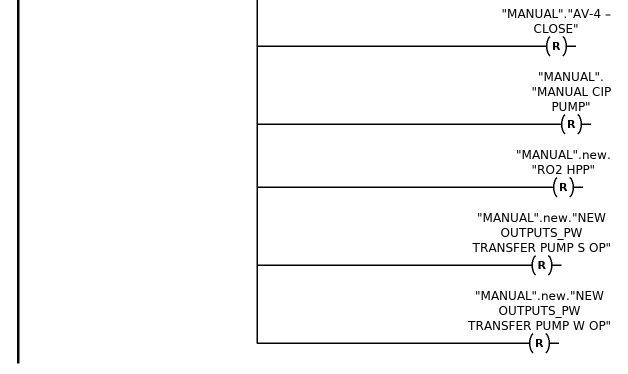
   RUNG wire#powerrail
      Contact( "AlwaysTRUE" )
      wire#w1
      { S7_Templates := "SrcType := Int" } NE_Contact(in1 := "Mode Select"."MFG MODE".BUFFER, in2 := 2)
      wire#w2
      R_Coil( "MANUAL"."MGF FEED PUMP WORKING" )
   END_RUNG
   RUNG wire#w1
      Contact( "INTERLOCK".ERROR )
   END_RUNG wire#w2
   RUNG wire#w2
      R_Coil( "MANUAL"."MFG FEED PUMP STANDBY" )
   END_RUNG
   RUNG wire#w2
      R_Coil( "MANUAL"."RO FEED PUMP WORKING" )
   END_RUNG
   RUNG wire#w2
      R_Coil( "MANUAL"."RO FEED PUMP STANDBY" )
   END_RUNG
   RUNG wire#w2
      R_Coil( "MANUAL"."RO HPP PUMP WORKING" )
   END_RUNG
   RUNG wire#w2
      R_Coil( "MANUAL"."RO HPP PUMP STANDBY" )
   END_RUNG
   RUNG wire#w2
      R_Coil( "MANUAL"."SMBS AGT-1" )
   END_RUNG
   RUNG wire#w2
      R_Coil( "MANUAL"."SALT TANK AGT-2" )
   END_RUNG
   RUNG wire#w2
      R_Coil( "MANUAL"."RO SMBS AGT-3" )
   END_RUNG
   RUNG wire#w2
      R_Coil( "MANUAL"."DP-1" )
   END_RUNG
   RUNG wire#w2
      R_Coil( "MANUAL"."DP-2" )
   END_RUNG
   RUNG wire#w2
      R_Coil( "MANUAL"."DP-3" )
   END_RUNG
   RUNG wire#w2
      R_Coil( "MANUAL"."DP-4" )
   END_RUNG
   RUNG wire#w2
      R_Coil( "MANUAL"."DP-5" )
   END_RUNG
   RUNG wire#w2
      R_Coil( "MANUAL"."DP-6" )
   END_RUNG
   RUNG wire#w2
      R_Coil( "MANUAL"."UV-1-DO" )
   END_RUNG
   RUNG wire#w2
      R_Coil( "MANUAL"."UV-2-DO" )
   END_RUNG
   RUNG wire#w2
      R_Coil( "MANUAL".HOOTER )
   END_RUNG
   RUNG wire#w2
      R_Coil( "MANUAL"."PSFV-1 – OPEN" )
   END_RUNG
   RUNG wire#w2
      R_Coil( "MANUAL"."PSFV-1 – CLOSE" )
   END_RUNG
   RUNG wire#w2
      R_Coil( "MANUAL"."PSFV-2 – OPEN" )
   END_RUNG
   RUNG wire#w2
      R_Coil( "MANUAL"."PSFV-2 – CLOSE" )
   END_RUNG
   RUNG wire#w2
      R_Coil( "MANUAL"."PSFV-3 – OPEN" )
   END_RUNG
   RUNG wire#w2
      R_Coil( "MANUAL"."PSFV-3 – CLOSE" )
   END_RUNG
   RUNG wire#w2
      R_Coil( "MANUAL"."PSFV-4 – OPEN" )
   END_RUNG
   RUNG wire#w2
      R_Coil( "MANUAL"."PSFV-4 – CLOSE" )
   END_RUNG
   RUNG wire#w2
      R_Coil( "MANUAL"."PSFV-5 – OPEN" )
   END_RUNG
   RUNG wire#w2
      R_Coil( "MANUAL"."PSFV-5 – CLOSE" )
   END_RUNG
   RUNG wire#w2
      R_Coil( "MANUAL"."PSFV-6 – OPEN" )
   END_RUNG
   RUNG wire#w2
      R_Coil( "MANUAL"."PSFV-6 – CLOSE" )
   END_RUNG
   RUNG wire#w2
      R_Coil( "MANUAL"."ACFV-1 – OPEN" )
   END_RUNG
   RUNG wire#w2
      R_Coil( "MANUAL"."ACFV-1 – CLOSE" )
   END_RUNG
   RUNG wire#w2
      R_Coil( "MANUAL"."ACFV-2 – OPEN" )
   END_RUNG
   RUNG wire#w2
      R_Coil( "MANUAL"."ACFV-2 – CLOSE" )
   END_RUNG
   RUNG wire#w2
      R_Coil( "MANUAL"."ACFV-3 – OPEN" )
   END_RUNG
   RUNG wire#w2
      R_Coil( "MANUAL"."ACFV-3 – CLOSE" )
   END_RUNG
   RUNG wire#w2
      R_Coil( "MANUAL"."ACFV-4 – OPEN" )
   END_RUNG
   RUNG wire#w2
      R_Coil( "MANUAL"."ACFV-4 - CLOSE" )
   END_RUNG
   RUNG wire#w2
      R_Coil( "MANUAL"."ACFV-5 – OPEN" )
   END_RUNG
   RUNG wire#w2
      R_Coil( "MANUAL"."ACFV-5 – CLOSE" )
   END_RUNG
   RUNG wire#w2
      R_Coil( "MANUAL"."ACFV-6 – OPEN" )
   END_RUNG
   RUNG wire#w2
      R_Coil( "MANUAL"."ACFV-6 – CLOSE" )
   END_RUNG
   RUNG wire#w2
      R_Coil( "MANUAL"."SFV-1 – OPEN" )
   END_RUNG
   RUNG wire#w2
      R_Coil( "MANUAL"."SFV-1 – CLOSE" )
   END_RUNG
   RUNG wire#w2
      R_Coil( "MANUAL"."SFV-2 – OPEN" )
   END_RUNG
   RUNG wire#w2
      R_Coil( "MANUAL"."SFV-2 – CLOSE" )
   END_RUNG
   RUNG wire#w2
      R_Coil( "MANUAL"."SFV-3 – OPEN" )
   END_RUNG
   RUNG wire#w2
      R_Coil( "MANUAL"."SFV-3 – CLOSE" )
   END_RUNG
   RUNG wire#w2
      R_Coil( "MANUAL"."SFV-4 – OPEN" )
   END_RUNG
   RUNG wire#w2
      R_Coil( "MANUAL"."SFV-4 – CLOSE" )
   END_RUNG
   RUNG wire#w2
      R_Coil( "MANUAL"."SFV-5 – OPEN" )
   END_RUNG
   RUNG wire#w2
      R_Coil( "MANUAL"."SFV-5 – CLOSE" )
   END_RUNG
   RUNG wire#w2
      R_Coil( "MANUAL"."SFV-6 – OPEN" )
   END_RUNG
   RUNG wire#w2
      R_Coil( "MANUAL"."SFV-6 – CLOSE" )
   END_RUNG
   RUNG wire#w2
      R_Coil( "MANUAL"."SFV-7 – OPEN" )
   END_RUNG
   RUNG wire#w2
      R_Coil( "MANUAL"."SFV-7 – CLOSE" )
   END_RUNG
   RUNG wire#w2
      R_Coil( "MANUAL"."SFV-8 – OPEN" )
   END_RUNG
   RUNG wire#w2
      R_Coil( "MANUAL"."SFV-8 – CLOSE" )
   END_RUNG
   RUNG wire#w2
      R_Coil( "MANUAL"."AV-1 – OPEN" )
   END_RUNG
   RUNG wire#w2
      R_Coil( "MANUAL"."AV-1 – CLOSE" )
   END_RUNG
   RUNG wire#w2
      R_Coil( "MANUAL"."AV-2 – OPEN" )
   END_RUNG
   RUNG wire#w2
      R_Coil( "MANUAL"."AV-2 – CLOSE" )
   END_RUNG
   RUNG wire#w2
      R_Coil( "MANUAL"."AV-3 – OPEN" )
   END_RUNG
   RUNG wire#w2
      R_Coil( "MANUAL"."AV-3 – CLOSE" )
   END_RUNG
   RUNG wire#w2
      R_Coil( "MANUAL"."AV-4 – OPEN" )
   END_RUNG
   RUNG wire#w2
      R_Coil( "MANUAL"."AV-4 – CLOSE" )
   END_RUNG
   RUNG wire#w2
      R_Coil( "MANUAL"."MANUAL CIP PUMP" )
   END_RUNG
   RUNG wire#w2
      R_Coil( "MANUAL".new."RO2 HPP" )
   END_RUNG
   RUNG wire#w2
      R_Coil( "MANUAL".new."NEW OUTPUTS_PW TRANSFER PUMP S OP" )
   END_RUNG
   RUNG wire#w2
      R_Coil( "MANUAL".new."NEW OUTPUTS_PW TRANSFER PUMP W OP" )
   END_RUNG
   // the same network as SCL:
   IF "AlwaysTRUE" AND (("Mode Select"."MFG MODE".BUFFER <> 2) OR "INTERLOCK".ERROR) THEN
       "MANUAL"."MGF FEED PUMP WORKING" := FALSE;
       "MANUAL"."MFG FEED PUMP STANDBY" := FALSE;
       "MANUAL"."RO FEED PUMP WORKING" := FALSE;
       "MANUAL"."RO FEED PUMP STANDBY" := FALSE;
       "MANUAL"."RO HPP PUMP WORKING" := FALSE;
       "MANUAL"."RO HPP PUMP STANDBY" := FALSE;
       "MANUAL"."SMBS AGT-1" := FALSE;
       "MANUAL"."SALT TANK AGT-2" := FALSE;
       "MANUAL"."RO SMBS AGT-3" := FALSE;
       "MANUAL"."DP-1" := FALSE;
       "MANUAL"."DP-2" := FALSE;
       "MANUAL"."DP-3" := FALSE;
       "MANUAL"."DP-4" := FALSE;
       "MANUAL"."DP-5" := FALSE;
       "MANUAL"."DP-6" := FALSE;
       "MANUAL"."UV-1-DO" := FALSE;
       "MANUAL"."UV-2-DO" := FALSE;
       "MANUAL".HOOTER := FALSE;
       "MANUAL"."PSFV-1 – OPEN" := FALSE;
       "MANUAL"."PSFV-1 – CLOSE" := FALSE;
       "MANUAL"."PSFV-2 – OPEN" := FALSE;
       "MANUAL"."PSFV-2 – CLOSE" := FALSE;
       "MANUAL"."PSFV-3 – OPEN" := FALSE;
       "MANUAL"."PSFV-3 – CLOSE" := FALSE;
       "MANUAL"."PSFV-4 – OPEN" := FALSE;
       "MANUAL"."PSFV-4 – CLOSE" := FALSE;
       "MANUAL"."PSFV-5 – OPEN" := FALSE;
       "MANUAL"."PSFV-5 – CLOSE" := FALSE;
       "MANUAL"."PSFV-6 – OPEN" := FALSE;
       "MANUAL"."PSFV-6 – CLOSE" := FALSE;
       "MANUAL"."ACFV-1 – OPEN" := FALSE;
       "MANUAL"."ACFV-1 – CLOSE" := FALSE;
       "MANUAL"."ACFV-2 – OPEN" := FALSE;
       "MANUAL"."ACFV-2 – CLOSE" := FALSE;
       "MANUAL"."ACFV-3 – OPEN" := FALSE;
       "MANUAL"."ACFV-3 – CLOSE" := FALSE;
       "MANUAL"."ACFV-4 – OPEN" := FALSE;
       "MANUAL"."ACFV-4 - CLOSE" := FALSE;
       "MANUAL"."ACFV-5 – OPEN" := FALSE;
       "MANUAL"."ACFV-5 – CLOSE" := FALSE;
       "MANUAL"."ACFV-6 – OPEN" := FALSE;
       "MANUAL"."ACFV-6 – CLOSE" := FALSE;
       "MANUAL"."SFV-1 – OPEN" := FALSE;
       "MANUAL"."SFV-1 – CLOSE" := FALSE;
       "MANUAL"."SFV-2 – OPEN" := FALSE;
       "MANUAL"."SFV-2 – CLOSE" := FALSE;
       "MANUAL"."SFV-3 – OPEN" := FALSE;
       "MANUAL"."SFV-3 – CLOSE" := FALSE;
       "MANUAL"."SFV-4 – OPEN" := FALSE;
       "MANUAL"."SFV-4 – CLOSE" := FALSE;
       "MANUAL"."SFV-5 – OPEN" := FALSE;
       "MANUAL"."SFV-5 – CLOSE" := FALSE;
       "MANUAL"."SFV-6 – OPEN" := FALSE;
       "MANUAL"."SFV-6 – CLOSE" := FALSE;
       "MANUAL"."SFV-7 – OPEN" := FALSE;
       "MANUAL"."SFV-7 – CLOSE" := FALSE;
       "MANUAL"."SFV-8 – OPEN" := FALSE;
       "MANUAL"."SFV-8 – CLOSE" := FALSE;
       "MANUAL"."AV-1 – OPEN" := FALSE;
       "MANUAL"."AV-1 – CLOSE" := FALSE;
       "MANUAL"."AV-2 – OPEN" := FALSE;
       "MANUAL"."AV-2 – CLOSE" := FALSE;
       "MANUAL"."AV-3 – OPEN" := FALSE;
       "MANUAL"."AV-3 – CLOSE" := FALSE;
       "MANUAL"."AV-4 – OPEN" := FALSE;
       "MANUAL"."AV-4 – CLOSE" := FALSE;
       "MANUAL"."MANUAL CIP PUMP" := FALSE;
       "MANUAL".new."RO2 HPP" := FALSE;
       "MANUAL".new."NEW OUTPUTS_PW TRANSFER PUMP S OP" := FALSE;
       "MANUAL".new."NEW OUTPUTS_PW TRANSFER PUMP W OP" := FALSE;
   END_IF;
END_REGION

REGION Network 3: TRANSFER PUMP WORKING & STANDBY
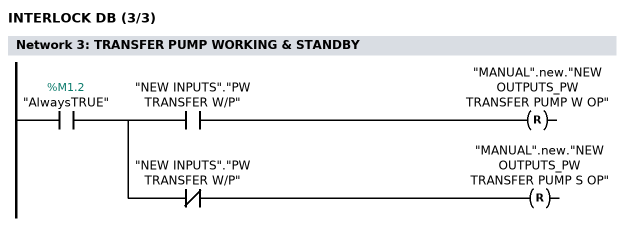
   RUNG wire#powerrail
      Contact( "AlwaysTRUE" )
      wire#w1
      Contact( "NEW INPUTS"."PW TRANSFER W/P" )
      R_Coil( "MANUAL".new."NEW OUTPUTS_PW TRANSFER PUMP W OP" )
   END_RUNG
   RUNG wire#w1
      I_Contact( "NEW INPUTS"."PW TRANSFER W/P" )
      R_Coil( "MANUAL".new."NEW OUTPUTS_PW TRANSFER PUMP S OP" )
   END_RUNG
   // the same network as SCL:
   IF "AlwaysTRUE" AND "NEW INPUTS"."PW TRANSFER W/P" THEN
       "MANUAL".new."NEW OUTPUTS_PW TRANSFER PUMP W OP" := FALSE;
   END_IF;
   IF "AlwaysTRUE" AND NOT "NEW INPUTS"."PW TRANSFER W/P" THEN
       "MANUAL".new."NEW OUTPUTS_PW TRANSFER PUMP S OP" := FALSE;
   END_IF;
END_REGION
END_FUNCTION

FUNCTION "SCALING" : Void   // FC3, LAD
{ S7_Optimized_Access := 'TRUE' }
// stored: SetENOAutomatically false
BEGIN

REGION Network 1: LT-1
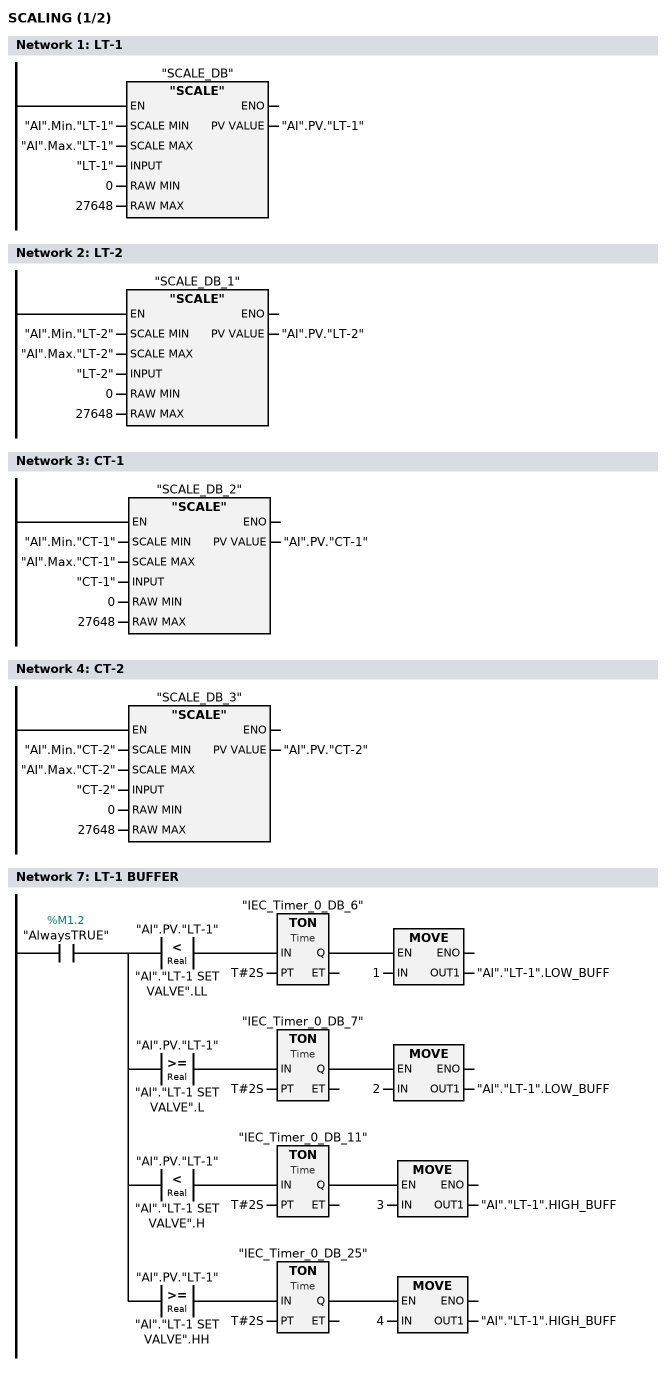
   RUNG wire#powerrail
      "SCALE_DB"("SCALE MIN" := "AI".Min."LT-1", "SCALE MAX" := "AI".Max."LT-1", INPUT := "LT-1", "RAW MIN" := 0, "RAW MAX" := 27648, "PV VALUE" => "AI".PV."LT-1")
   END_RUNG
   // the same network as SCL:
   "SCALE_DB"("SCALE MIN" := "AI".Min."LT-1",   // "SCALE"
              "SCALE MAX" := "AI".Max."LT-1",
              INPUT := "LT-1",
              "RAW MIN" := 0,
              "RAW MAX" := 27648,
              "PV VALUE" => "AI".PV."LT-1");
END_REGION

REGION Network 2: LT-2
   RUNG wire#powerrail
      "SCALE_DB_1"("SCALE MIN" := "AI".Min."LT-2", "SCALE MAX" := "AI".Max."LT-2", INPUT := "LT-2", "RAW MIN" := 0, "RAW MAX" := 27648, "PV VALUE" => "AI".PV."LT-2")
   END_RUNG
   // the same network as SCL:
   "SCALE_DB_1"("SCALE MIN" := "AI".Min."LT-2",   // "SCALE"
                "SCALE MAX" := "AI".Max."LT-2",
                INPUT := "LT-2",
                "RAW MIN" := 0,
                "RAW MAX" := 27648,
                "PV VALUE" => "AI".PV."LT-2");
END_REGION

REGION Network 3: CT-1
   RUNG wire#powerrail
      "SCALE_DB_2"("SCALE MIN" := "AI".Min."CT-1", "SCALE MAX" := "AI".Max."CT-1", INPUT := "CT-1", "RAW MIN" := 0, "RAW MAX" := 27648, "PV VALUE" => "AI".PV."CT-1")
   END_RUNG
   // the same network as SCL:
   "SCALE_DB_2"("SCALE MIN" := "AI".Min."CT-1",   // "SCALE"
                "SCALE MAX" := "AI".Max."CT-1",
                INPUT := "CT-1",
                "RAW MIN" := 0,
                "RAW MAX" := 27648,
                "PV VALUE" => "AI".PV."CT-1");
END_REGION

REGION Network 4: CT-2
   RUNG wire#powerrail
      "SCALE_DB_3"("SCALE MIN" := "AI".Min."CT-2", "SCALE MAX" := "AI".Max."CT-2", INPUT := "CT-2", "RAW MIN" := 0, "RAW MAX" := 27648, "PV VALUE" => "AI".PV."CT-2")
   END_RUNG
   // the same network as SCL:
   "SCALE_DB_3"("SCALE MIN" := "AI".Min."CT-2",   // "SCALE"
                "SCALE MAX" := "AI".Max."CT-2",
                INPUT := "CT-2",
                "RAW MIN" := 0,
                "RAW MAX" := 27648,
                "PV VALUE" => "AI".PV."CT-2");
END_REGION

REGION Network 7: LT-1 BUFFER
   RUNG wire#powerrail
      Contact( "AlwaysTRUE" )
      wire#w1
      { S7_Templates := "SrcType := Real" } LT_Contact(in1 := "AI".PV."LT-1", in2 := "AI"."LT-1 SET VALVE".LL)
      { S7_Templates := "time_type := Time" } "IEC_Timer_0_DB_6".TON(pt := T#2S, et =>)
      Move(in := 1, out1 => "AI"."LT-1".LOW_BUFF)
   END_RUNG
   RUNG wire#w1
      { S7_Templates := "SrcType := Real" } GE_Contact(in1 := "AI".PV."LT-1", in2 := "AI"."LT-1 SET VALVE".L)
      { S7_Templates := "time_type := Time" } "IEC_Timer_0_DB_7".TON(pt := T#2S, et =>)
      Move(in := 2, out1 => "AI"."LT-1".LOW_BUFF)
   END_RUNG
   RUNG wire#w1
      { S7_Templates := "SrcType := Real" } LT_Contact(in1 := "AI".PV."LT-1", in2 := "AI"."LT-1 SET VALVE".H)
      { S7_Templates := "time_type := Time" } "IEC_Timer_0_DB_11".TON(pt := T#2S, et =>)
      Move(in := 3, out1 => "AI"."LT-1".HIGH_BUFF)
   END_RUNG
   RUNG wire#w1
      { S7_Templates := "SrcType := Real" } GE_Contact(in1 := "AI".PV."LT-1", in2 := "AI"."LT-1 SET VALVE".HH)
      { S7_Templates := "time_type := Time" } "IEC_Timer_0_DB_25".TON(pt := T#2S, et =>)
      Move(in := 4, out1 => "AI"."LT-1".HIGH_BUFF)
   END_RUNG
   // the same network as SCL:
   "IEC_Timer_0_DB_6".TON(IN := "AlwaysTRUE" AND ("AI".PV."LT-1" < "AI"."LT-1 SET VALVE".LL), PT := T#2S);
   IF "IEC_Timer_0_DB_6".Q THEN "AI"."LT-1".LOW_BUFF := 1; END_IF;
   "IEC_Timer_0_DB_7".TON(IN := "AlwaysTRUE" AND ("AI".PV."LT-1" >= "AI"."LT-1 SET VALVE".L), PT := T#2S);
   IF "IEC_Timer_0_DB_7".Q THEN "AI"."LT-1".LOW_BUFF := 2; END_IF;
   "IEC_Timer_0_DB_11".TON(IN := "AlwaysTRUE" AND ("AI".PV."LT-1" < "AI"."LT-1 SET VALVE".H), PT := T#2S);
   IF "IEC_Timer_0_DB_11".Q THEN "AI"."LT-1".HIGH_BUFF := 3; END_IF;
   "IEC_Timer_0_DB_25".TON(IN := "AlwaysTRUE" AND ("AI".PV."LT-1" >= "AI"."LT-1 SET VALVE".HH), PT := T#2S);
   IF "IEC_Timer_0_DB_25".Q THEN "AI"."LT-1".HIGH_BUFF := 4; END_IF;
END_REGION

REGION Network 8: LT-2 BUFFER
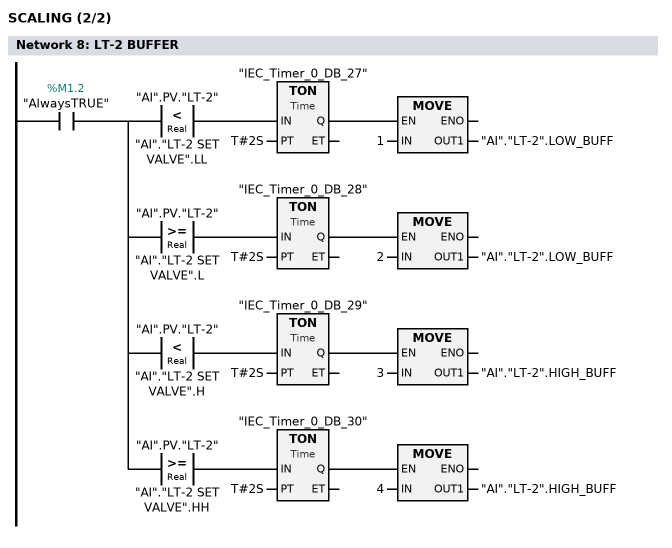
   RUNG wire#powerrail
      Contact( "AlwaysTRUE" )
      wire#w1
      { S7_Templates := "SrcType := Real" } LT_Contact(in1 := "AI".PV."LT-2", in2 := "AI"."LT-2 SET VALVE".LL)
      { S7_Templates := "time_type := Time" } "IEC_Timer_0_DB_27".TON(pt := T#2S, et =>)
      Move(in := 1, out1 => "AI"."LT-2".LOW_BUFF)
   END_RUNG
   RUNG wire#w1
      { S7_Templates := "SrcType := Real" } GE_Contact(in1 := "AI".PV."LT-2", in2 := "AI"."LT-2 SET VALVE".L)
      { S7_Templates := "time_type := Time" } "IEC_Timer_0_DB_28".TON(pt := T#2S, et =>)
      Move(in := 2, out1 => "AI"."LT-2".LOW_BUFF)
   END_RUNG
   RUNG wire#w1
      { S7_Templates := "SrcType := Real" } LT_Contact(in1 := "AI".PV."LT-2", in2 := "AI"."LT-2 SET VALVE".H)
      { S7_Templates := "time_type := Time" } "IEC_Timer_0_DB_29".TON(pt := T#2S, et =>)
      Move(in := 3, out1 => "AI"."LT-2".HIGH_BUFF)
   END_RUNG
   RUNG wire#w1
      { S7_Templates := "SrcType := Real" } GE_Contact(in1 := "AI".PV."LT-2", in2 := "AI"."LT-2 SET VALVE".HH)
      { S7_Templates := "time_type := Time" } "IEC_Timer_0_DB_30".TON(pt := T#2S, et =>)
      Move(in := 4, out1 => "AI"."LT-2".HIGH_BUFF)
   END_RUNG
   // the same network as SCL:
   "IEC_Timer_0_DB_27".TON(IN := "AlwaysTRUE" AND ("AI".PV."LT-2" < "AI"."LT-2 SET VALVE".LL), PT := T#2S);
   IF "IEC_Timer_0_DB_27".Q THEN "AI"."LT-2".LOW_BUFF := 1; END_IF;
   "IEC_Timer_0_DB_28".TON(IN := "AlwaysTRUE" AND ("AI".PV."LT-2" >= "AI"."LT-2 SET VALVE".L), PT := T#2S);
   IF "IEC_Timer_0_DB_28".Q THEN "AI"."LT-2".LOW_BUFF := 2; END_IF;
   "IEC_Timer_0_DB_29".TON(IN := "AlwaysTRUE" AND ("AI".PV."LT-2" < "AI"."LT-2 SET VALVE".H), PT := T#2S);
   IF "IEC_Timer_0_DB_29".Q THEN "AI"."LT-2".HIGH_BUFF := 3; END_IF;
   "IEC_Timer_0_DB_30".TON(IN := "AlwaysTRUE" AND ("AI".PV."LT-2" >= "AI"."LT-2 SET VALVE".HH), PT := T#2S);
   IF "IEC_Timer_0_DB_30".Q THEN "AI"."LT-2".HIGH_BUFF := 4; END_IF;
END_REGION
END_FUNCTION

FUNCTION_BLOCK "SCALE"   // FB4, LAD
{ S7_Optimized_Access := 'TRUE' }
// stored: MemoryReserve 100, SetENOAutomatically false
   VAR_INPUT
      "SCALE MIN" : Real;
      "SCALE MAX" : Real;
      INPUT : Int;
      "RAW MIN" : Int;
      "RAW MAX" : Int;
   END_VAR
   VAR_OUTPUT
      "PV VALUE" : Real;
   END_VAR
   VAR_TEMP
      NORMX : Real;
   END_VAR
BEGIN

REGION Network 1
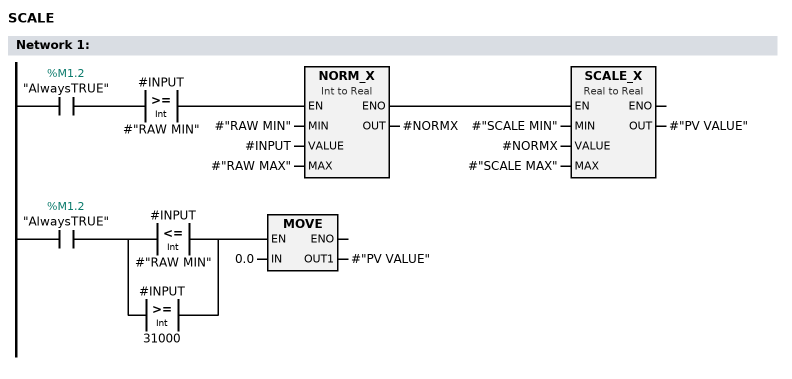
   RUNG wire#powerrail
      Contact( "AlwaysTRUE" )
      { S7_Templates := "SrcType := Int" } GE_Contact(in1 := #INPUT, in2 := #"RAW MIN")
      { S7_Templates := "[SrcType := Int, DestType := Real]" } Normalize(min := #"RAW MIN", value := #INPUT, max := #"RAW MAX", out => #NORMX)
      { S7_Templates := "[SrcType := Real, DestType := Real]" } Scale(min := #"SCALE MIN", value := #NORMX, max := #"SCALE MAX", out => #"PV VALUE")
   END_RUNG
   RUNG wire#powerrail
      Contact( "AlwaysTRUE" )
      wire#w1
      { S7_Templates := "SrcType := Int" } LE_Contact(in1 := #INPUT, in2 := #"RAW MIN")
      wire#w2
      Move(in := 0.0, out1 => #"PV VALUE")
   END_RUNG
   RUNG wire#w1
      { S7_Templates := "SrcType := Int" } GE_Contact(in1 := #INPUT, in2 := 31000)
   END_RUNG wire#w2
   // the same network as SCL:
   IF "AlwaysTRUE" AND (#INPUT >= #"RAW MIN") THEN
       #NORMX := NORM_X(MIN := #"RAW MIN", VALUE := #INPUT, MAX := #"RAW MAX");
       #"PV VALUE" := SCALE_X(MIN := #"SCALE MIN", VALUE := #NORMX, MAX := #"SCALE MAX");
   END_IF;
   IF "AlwaysTRUE" AND ((#INPUT <= #"RAW MIN") OR (#INPUT >= 31000)) THEN #"PV VALUE" := 0.0; END_IF;
END_REGION
END_FUNCTION_BLOCK

FUNCTION "ALARMS" : Void   // FC16, LAD
{ S7_Optimized_Access := 'TRUE' }
// stored: SetENOAutomatically false
   VAR_TEMP   // added for the SCL form of the ladder/FBD networks
      _w1 : Bool;
   END_VAR
BEGIN

REGION Network 1: EMG ALARM
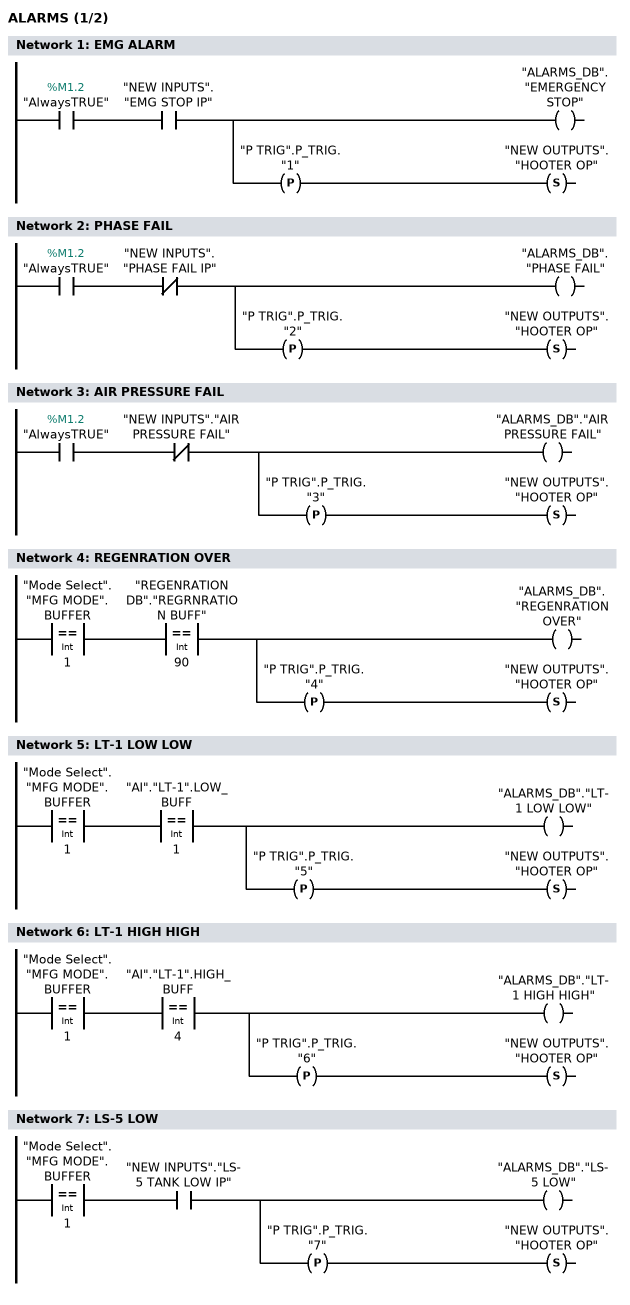
   RUNG wire#powerrail
      Contact( "AlwaysTRUE" )
      Contact( "NEW INPUTS"."EMG STOP IP" )
      wire#w1
      Coil( "ALARMS_DB"."EMERGENCY STOP" )
   END_RUNG
   RUNG wire#w1
      P_Trig( "P TRIG".P_TRIG."1" )
      S_Coil( "NEW OUTPUTS"."HOOTER OP" )
   END_RUNG
   // the same network as SCL:
   "ALARMS_DB"."EMERGENCY STOP" := "AlwaysTRUE" AND "NEW INPUTS"."EMG STOP IP";
   #_w1 := "ALARMS_DB"."EMERGENCY STOP" AND NOT "P TRIG".P_TRIG."1";   // rising edge
   "P TRIG".P_TRIG."1" := "ALARMS_DB"."EMERGENCY STOP";
   IF #_w1 THEN "NEW OUTPUTS"."HOOTER OP" := TRUE; END_IF;
END_REGION

REGION Network 2: PHASE FAIL
   RUNG wire#powerrail
      Contact( "AlwaysTRUE" )
      I_Contact( "NEW INPUTS"."PHASE FAIL IP" )
      wire#w1
      Coil( "ALARMS_DB"."PHASE FAIL" )
   END_RUNG
   RUNG wire#w1
      P_Trig( "P TRIG".P_TRIG."2" )
      S_Coil( "NEW OUTPUTS"."HOOTER OP" )
   END_RUNG
   // the same network as SCL:
   "ALARMS_DB"."PHASE FAIL" := "AlwaysTRUE" AND NOT "NEW INPUTS"."PHASE FAIL IP";
   #_w1 := "ALARMS_DB"."PHASE FAIL" AND NOT "P TRIG".P_TRIG."2";   // rising edge
   "P TRIG".P_TRIG."2" := "ALARMS_DB"."PHASE FAIL";
   IF #_w1 THEN "NEW OUTPUTS"."HOOTER OP" := TRUE; END_IF;
END_REGION

REGION Network 3: AIR PRESSURE FAIL
   RUNG wire#powerrail
      Contact( "AlwaysTRUE" )
      I_Contact( "NEW INPUTS"."AIR PRESSURE FAIL" )
      wire#w1
      Coil( "ALARMS_DB"."AIR PRESSURE FAIL" )
   END_RUNG
   RUNG wire#w1
      P_Trig( "P TRIG".P_TRIG."3" )
      S_Coil( "NEW OUTPUTS"."HOOTER OP" )
   END_RUNG
   // the same network as SCL:
   "ALARMS_DB"."AIR PRESSURE FAIL" := "AlwaysTRUE" AND NOT "NEW INPUTS"."AIR PRESSURE FAIL";
   #_w1 := "ALARMS_DB"."AIR PRESSURE FAIL" AND NOT "P TRIG".P_TRIG."3";   // rising edge
   "P TRIG".P_TRIG."3" := "ALARMS_DB"."AIR PRESSURE FAIL";
   IF #_w1 THEN "NEW OUTPUTS"."HOOTER OP" := TRUE; END_IF;
END_REGION

REGION Network 4: REGENRATION OVER
   RUNG wire#powerrail
      { S7_Templates := "SrcType := Int" } EQ_Contact(in1 := "Mode Select"."MFG MODE".BUFFER, in2 := 1)
      { S7_Templates := "SrcType := Int" } EQ_Contact(in1 := "REGENRATION DB"."REGRNRATION BUFF", in2 := 90)
      wire#w1
      Coil( "ALARMS_DB"."REGENRATION OVER" )
   END_RUNG
   RUNG wire#w1
      P_Trig( "P TRIG".P_TRIG."4" )
      S_Coil( "NEW OUTPUTS"."HOOTER OP" )
   END_RUNG
   // the same network as SCL:
   "ALARMS_DB"."REGENRATION OVER" := ("Mode Select"."MFG MODE".BUFFER = 1) AND ("REGENRATION DB"."REGRNRATION BUFF" = 90);
   #_w1 := "ALARMS_DB"."REGENRATION OVER" AND NOT "P TRIG".P_TRIG."4";   // rising edge
   "P TRIG".P_TRIG."4" := "ALARMS_DB"."REGENRATION OVER";
   IF #_w1 THEN "NEW OUTPUTS"."HOOTER OP" := TRUE; END_IF;
END_REGION

REGION Network 5: LT-1 LOW LOW
   RUNG wire#powerrail
      { S7_Templates := "SrcType := Int" } EQ_Contact(in1 := "Mode Select"."MFG MODE".BUFFER, in2 := 1)
      { S7_Templates := "SrcType := Int" } EQ_Contact(in1 := "AI"."LT-1".LOW_BUFF, in2 := 1)
      wire#w1
      Coil( "ALARMS_DB"."LT-1 LOW LOW" )
   END_RUNG
   RUNG wire#w1
      P_Trig( "P TRIG".P_TRIG."5" )
      S_Coil( "NEW OUTPUTS"."HOOTER OP" )
   END_RUNG
   // the same network as SCL:
   "ALARMS_DB"."LT-1 LOW LOW" := ("Mode Select"."MFG MODE".BUFFER = 1) AND ("AI"."LT-1".LOW_BUFF = 1);
   #_w1 := "ALARMS_DB"."LT-1 LOW LOW" AND NOT "P TRIG".P_TRIG."5";   // rising edge
   "P TRIG".P_TRIG."5" := "ALARMS_DB"."LT-1 LOW LOW";
   IF #_w1 THEN "NEW OUTPUTS"."HOOTER OP" := TRUE; END_IF;
END_REGION

REGION Network 6: LT-1 HIGH HIGH
   RUNG wire#powerrail
      { S7_Templates := "SrcType := Int" } EQ_Contact(in1 := "Mode Select"."MFG MODE".BUFFER, in2 := 1)
      { S7_Templates := "SrcType := Int" } EQ_Contact(in1 := "AI"."LT-1".HIGH_BUFF, in2 := 4)
      wire#w1
      Coil( "ALARMS_DB"."LT-1 HIGH HIGH" )
   END_RUNG
   RUNG wire#w1
      P_Trig( "P TRIG".P_TRIG."6" )
      S_Coil( "NEW OUTPUTS"."HOOTER OP" )
   END_RUNG
   // the same network as SCL:
   "ALARMS_DB"."LT-1 HIGH HIGH" := ("Mode Select"."MFG MODE".BUFFER = 1) AND ("AI"."LT-1".HIGH_BUFF = 4);
   #_w1 := "ALARMS_DB"."LT-1 HIGH HIGH" AND NOT "P TRIG".P_TRIG."6";   // rising edge
   "P TRIG".P_TRIG."6" := "ALARMS_DB"."LT-1 HIGH HIGH";
   IF #_w1 THEN "NEW OUTPUTS"."HOOTER OP" := TRUE; END_IF;
END_REGION

REGION Network 7: LS-5 LOW
   RUNG wire#powerrail
      { S7_Templates := "SrcType := Int" } EQ_Contact(in1 := "Mode Select"."MFG MODE".BUFFER, in2 := 1)
      Contact( "NEW INPUTS"."LS-5 TANK LOW IP" )
      wire#w1
      Coil( "ALARMS_DB"."LS-5 LOW" )
   END_RUNG
   RUNG wire#w1
      P_Trig( "P TRIG".P_TRIG."7" )
      S_Coil( "NEW OUTPUTS"."HOOTER OP" )
   END_RUNG
   // the same network as SCL:
   "ALARMS_DB"."LS-5 LOW" := ("Mode Select"."MFG MODE".BUFFER = 1) AND "NEW INPUTS"."LS-5 TANK LOW IP";
   #_w1 := "ALARMS_DB"."LS-5 LOW" AND NOT "P TRIG".P_TRIG."7";   // rising edge
   "P TRIG".P_TRIG."7" := "ALARMS_DB"."LS-5 LOW";
   IF #_w1 THEN "NEW OUTPUTS"."HOOTER OP" := TRUE; END_IF;
END_REGION

REGION Network 8: PS-1 LOW
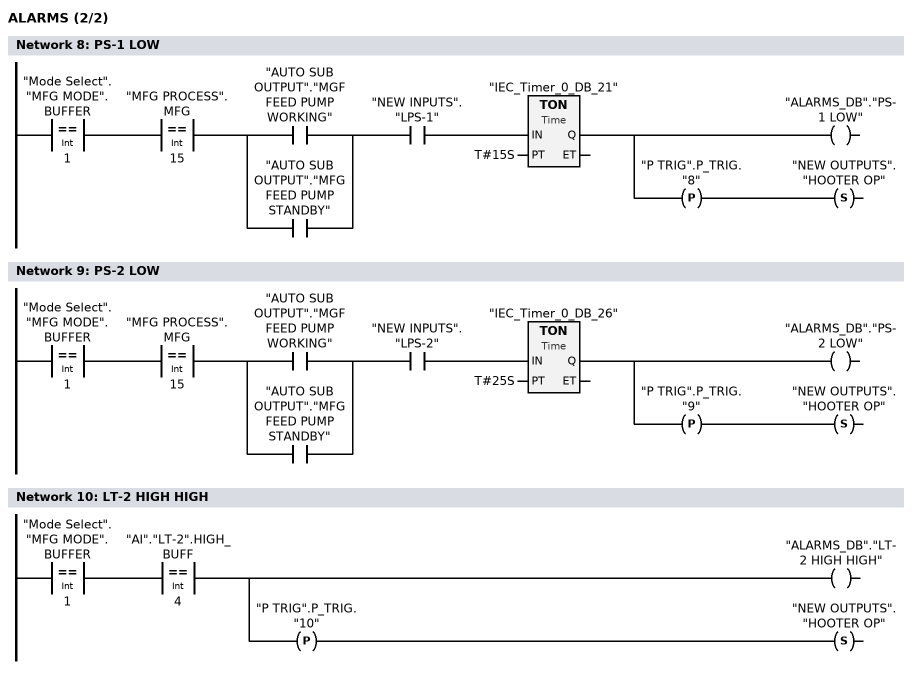
   RUNG wire#powerrail
      { S7_Templates := "SrcType := Int" } EQ_Contact(in1 := "Mode Select"."MFG MODE".BUFFER, in2 := 1)
      { S7_Templates := "SrcType := Int" } EQ_Contact(in1 := "MFG PROCESS".MFG, in2 := 15)
      wire#w1
      Contact( "AUTO SUB OUTPUT"."MGF FEED PUMP WORKING" )
      wire#w2
      Contact( "NEW INPUTS"."LPS-1" )
      { S7_Templates := "time_type := Time" } "IEC_Timer_0_DB_21".TON(pt := T#15S, et =>)
      wire#w3
      Coil( "ALARMS_DB"."PS-1 LOW" )
   END_RUNG
   RUNG wire#w1
      Contact( "AUTO SUB OUTPUT"."MFG FEED PUMP STANDBY" )
   END_RUNG wire#w2
   RUNG wire#w3
      P_Trig( "P TRIG".P_TRIG."8" )
      S_Coil( "NEW OUTPUTS"."HOOTER OP" )
   END_RUNG
   // the same network as SCL:
   "IEC_Timer_0_DB_21".TON(IN := ("Mode Select"."MFG MODE".BUFFER = 1) AND ("MFG PROCESS".MFG = 15) AND ("AUTO SUB OUTPUT"."MGF FEED PUMP WORKING" OR "AUTO SUB OUTPUT"."MFG FEED PUMP STANDBY") AND "NEW INPUTS"."LPS-1",
                           PT := T#15S);
   "ALARMS_DB"."PS-1 LOW" := "IEC_Timer_0_DB_21".Q;
   #_w1 := "IEC_Timer_0_DB_21".Q AND NOT "P TRIG".P_TRIG."8";   // rising edge
   "P TRIG".P_TRIG."8" := "IEC_Timer_0_DB_21".Q;
   IF #_w1 THEN "NEW OUTPUTS"."HOOTER OP" := TRUE; END_IF;
END_REGION

REGION Network 9: PS-2 LOW
   RUNG wire#powerrail
      { S7_Templates := "SrcType := Int" } EQ_Contact(in1 := "Mode Select"."MFG MODE".BUFFER, in2 := 1)
      { S7_Templates := "SrcType := Int" } EQ_Contact(in1 := "MFG PROCESS".MFG, in2 := 15)
      wire#w1
      Contact( "AUTO SUB OUTPUT"."MGF FEED PUMP WORKING" )
      wire#w2
      Contact( "NEW INPUTS"."LPS-2" )
      { S7_Templates := "time_type := Time" } "IEC_Timer_0_DB_26".TON(pt := T#25S, et =>)
      wire#w3
      Coil( "ALARMS_DB"."PS-2 LOW" )
   END_RUNG
   RUNG wire#w1
      Contact( "AUTO SUB OUTPUT"."MFG FEED PUMP STANDBY" )
   END_RUNG wire#w2
   RUNG wire#w3
      P_Trig( "P TRIG".P_TRIG."9" )
      S_Coil( "NEW OUTPUTS"."HOOTER OP" )
   END_RUNG
   // the same network as SCL:
   "IEC_Timer_0_DB_26".TON(IN := ("Mode Select"."MFG MODE".BUFFER = 1) AND ("MFG PROCESS".MFG = 15) AND ("AUTO SUB OUTPUT"."MGF FEED PUMP WORKING" OR "AUTO SUB OUTPUT"."MFG FEED PUMP STANDBY") AND "NEW INPUTS"."LPS-2",
                           PT := T#25S);
   "ALARMS_DB"."PS-2 LOW" := "IEC_Timer_0_DB_26".Q;
   #_w1 := "IEC_Timer_0_DB_26".Q AND NOT "P TRIG".P_TRIG."9";   // rising edge
   "P TRIG".P_TRIG."9" := "IEC_Timer_0_DB_26".Q;
   IF #_w1 THEN "NEW OUTPUTS"."HOOTER OP" := TRUE; END_IF;
END_REGION

REGION Network 10: LT-2 HIGH HIGH
   RUNG wire#powerrail
      { S7_Templates := "SrcType := Int" } EQ_Contact(in1 := "Mode Select"."MFG MODE".BUFFER, in2 := 1)
      { S7_Templates := "SrcType := Int" } EQ_Contact(in1 := "AI"."LT-2".HIGH_BUFF, in2 := 4)
      wire#w1
      Coil( "ALARMS_DB"."LT-2 HIGH HIGH" )
   END_RUNG
   RUNG wire#w1
      P_Trig( "P TRIG".P_TRIG."10" )
      S_Coil( "NEW OUTPUTS"."HOOTER OP" )
   END_RUNG
   // the same network as SCL:
   "ALARMS_DB"."LT-2 HIGH HIGH" := ("Mode Select"."MFG MODE".BUFFER = 1) AND ("AI"."LT-2".HIGH_BUFF = 4);
   #_w1 := "ALARMS_DB"."LT-2 HIGH HIGH" AND NOT "P TRIG".P_TRIG."10";   // rising edge
   "P TRIG".P_TRIG."10" := "ALARMS_DB"."LT-2 HIGH HIGH";
   IF #_w1 THEN "NEW OUTPUTS"."HOOTER OP" := TRUE; END_IF;
END_REGION
END_FUNCTION

FUNCTION "24 HOUR TIMER" : Void   // FC12, LAD
{ S7_Optimized_Access := 'TRUE' }
// stored: SetENOAutomatically false
   VAR_TEMP   // added for the SCL form of the ladder/FBD networks
      _w1 : Bool;
   END_VAR
BEGIN

REGION Network 1: 24 HOUR_TIMER
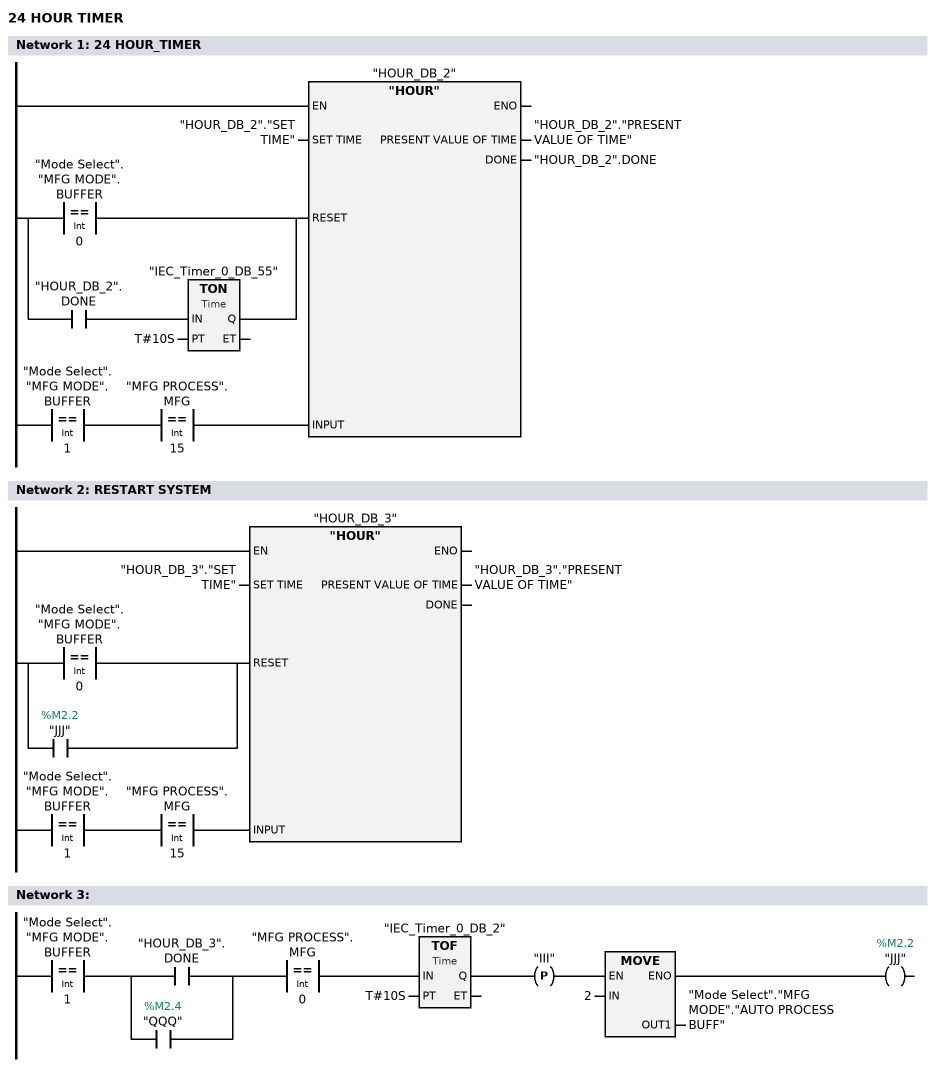
   RUNG wire#powerrail
      "HOUR_DB_2"(RESET := wire#w1, INPUT := wire#w2, "SET TIME" := "HOUR_DB_2"."SET TIME", "PRESENT VALUE OF TIME" => "HOUR_DB_2"."PRESENT VALUE OF TIME", DONE => "HOUR_DB_2".DONE)
   END_RUNG
   RUNG wire#powerrail
      { S7_Templates := "SrcType := Int" } EQ_Contact(in1 := "Mode Select"."MFG MODE".BUFFER, in2 := 0)
   END_RUNG wire#w1
   RUNG wire#powerrail
      Contact( "HOUR_DB_2".DONE )
      { S7_Templates := "time_type := Time" } "IEC_Timer_0_DB_55".TON(pt := T#10S, et =>)
   END_RUNG wire#w1
   RUNG wire#powerrail
      { S7_Templates := "SrcType := Int" } EQ_Contact(in1 := "Mode Select"."MFG MODE".BUFFER, in2 := 1)
      { S7_Templates := "SrcType := Int" } EQ_Contact(in1 := "MFG PROCESS".MFG, in2 := 15)
   END_RUNG wire#w2
   // the same network as SCL:
   "IEC_Timer_0_DB_55".TON(IN := "HOUR_DB_2".DONE, PT := T#10S);
   "HOUR_DB_2"("SET TIME" := "HOUR_DB_2"."SET TIME",   // "HOUR"
               RESET := ("Mode Select"."MFG MODE".BUFFER = 0) OR "IEC_Timer_0_DB_55".Q,
               INPUT := ("Mode Select"."MFG MODE".BUFFER = 1) AND ("MFG PROCESS".MFG = 15),
               "PRESENT VALUE OF TIME" => "HOUR_DB_2"."PRESENT VALUE OF TIME",
               DONE => "HOUR_DB_2".DONE);
END_REGION

REGION Network 2: RESTART SYSTEM
   RUNG wire#powerrail
      "HOUR_DB_3"(RESET := wire#w1, INPUT := wire#w2, "SET TIME" := "HOUR_DB_3"."SET TIME", "PRESENT VALUE OF TIME" => "HOUR_DB_3"."PRESENT VALUE OF TIME", DONE =>)
   END_RUNG
   RUNG wire#powerrail
      { S7_Templates := "SrcType := Int" } EQ_Contact(in1 := "Mode Select"."MFG MODE".BUFFER, in2 := 0)
   END_RUNG wire#w1
   RUNG wire#powerrail
      Contact( "JJJ" )
   END_RUNG wire#w1
   RUNG wire#powerrail
      { S7_Templates := "SrcType := Int" } EQ_Contact(in1 := "Mode Select"."MFG MODE".BUFFER, in2 := 1)
      { S7_Templates := "SrcType := Int" } EQ_Contact(in1 := "MFG PROCESS".MFG, in2 := 15)
   END_RUNG wire#w2
   // the same network as SCL:
   "HOUR_DB_3"("SET TIME" := "HOUR_DB_3"."SET TIME",   // "HOUR"
               RESET := ("Mode Select"."MFG MODE".BUFFER = 0) OR "JJJ",
               INPUT := ("Mode Select"."MFG MODE".BUFFER = 1) AND ("MFG PROCESS".MFG = 15),
               "PRESENT VALUE OF TIME" => "HOUR_DB_3"."PRESENT VALUE OF TIME");
END_REGION

REGION Network 3
   RUNG wire#powerrail
      { S7_Templates := "SrcType := Int" } EQ_Contact(in1 := "Mode Select"."MFG MODE".BUFFER, in2 := 1)
      wire#w1
      Contact( "HOUR_DB_3".DONE )
      wire#w2
      { S7_Templates := "SrcType := Int" } EQ_Contact(in1 := "MFG PROCESS".MFG, in2 := 0)
      { S7_Templates := "time_type := Time" } "IEC_Timer_0_DB_2".TOF(pt := T#10S, et =>)
      P_Trig( "III" )
      Move(in := 2, out1 => "Mode Select"."MFG MODE"."AUTO PROCESS BUFF")
      Coil( "JJJ" )
   END_RUNG
   RUNG wire#w1
      Contact( "QQQ" )
   END_RUNG wire#w2
   // the same network as SCL:
   "IEC_Timer_0_DB_2".TOF(IN := ("Mode Select"."MFG MODE".BUFFER = 1) AND ("HOUR_DB_3".DONE OR "QQQ") AND ("MFG PROCESS".MFG = 0),
                          PT := T#10S);
   #_w1 := "IEC_Timer_0_DB_2".Q AND NOT "III";   // rising edge
   "III" := "IEC_Timer_0_DB_2".Q;
   IF #_w1 THEN "Mode Select"."MFG MODE"."AUTO PROCESS BUFF" := 2; END_IF;
   "JJJ" := #_w1;
END_REGION
END_FUNCTION

FUNCTION_BLOCK "HOUR"   // FB2, LAD
{ S7_Optimized_Access := 'TRUE' }
// stored: MemoryReserve 100, SetENOAutomatically false
   VAR_INPUT
      "SET TIME" : Int;
      RESET : Bool;
      INPUT : Bool;
   END_VAR
   VAR_OUTPUT
      "PRESENT VALUE OF TIME" : Int;
      DONE : Bool;
   END_VAR
   VAR
      "TIMER 1" { S7_SetPoint := 'True'} : IEC_TIMER;
   END_VAR
   VAR RETAIN
      "COUNTER1 2" { S7_SetPoint := 'True'} : IEC_COUNTER;
      "COUNTER1 1" { S7_SetPoint := 'True'} : IEC_COUNTER;
   END_VAR
   VAR
      BIT { ExternalAccessible := 'False'; ExternalVisible := 'False'; ExternalWritable := 'False'} : Bool;
   END_VAR
   VAR_TEMP   // added for the SCL form of the ladder/FBD networks
      _w1 : Bool;
      _w2 : Bool;
   END_VAR
BEGIN

REGION Network 1
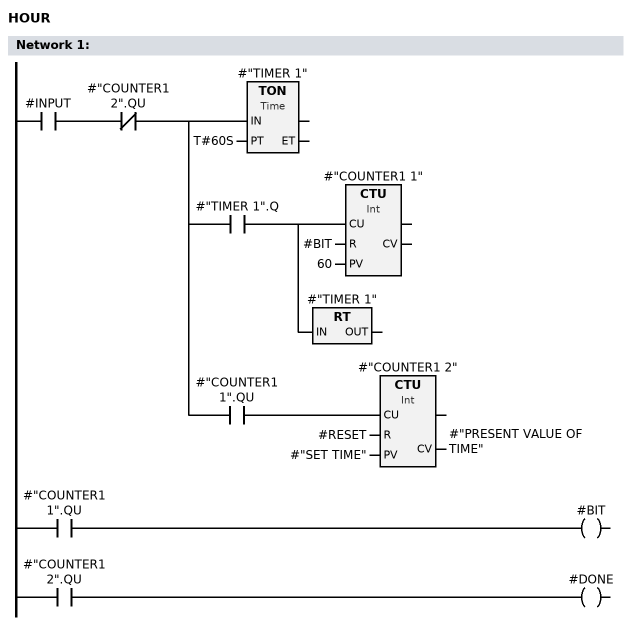
   RUNG wire#powerrail
      Contact( #INPUT )
      I_Contact( #"COUNTER1 2".QU )
      wire#w1
      { S7_Templates := "time_type := Time" } #"TIMER 1".TON(pt := T#60S, et =>)
   END_RUNG
   RUNG wire#w1
      Contact( #"TIMER 1".Q )
      wire#w2
      { S7_Templates := "value_type := Int" } #"COUNTER1 1".CTU(r := #BIT, pv := 60, cv =>)
   END_RUNG
   RUNG wire#w2
      RT_Coil( #"TIMER 1" )
   END_RUNG
   RUNG wire#w1
      Contact( #"COUNTER1 1".QU )
      { S7_Templates := "value_type := Int" } #"COUNTER1 2".CTU(r := #RESET, pv := #"SET TIME", cv => #"PRESENT VALUE OF TIME")
   END_RUNG
   RUNG wire#powerrail
      Contact( #"COUNTER1 1".QU )
      Coil( #BIT )
   END_RUNG
   RUNG wire#powerrail
      Contact( #"COUNTER1 2".QU )
      Coil( #DONE )
   END_RUNG
   // the same network as SCL:
   #_w1 := #INPUT AND NOT #"COUNTER1 2".QU;
   #"TIMER 1".TON(IN := #_w1, PT := T#60S);
   #_w2 := #_w1 AND #"TIMER 1".Q;
   #"COUNTER1 1".CTU(CU := #_w2, R := #BIT, PV := 60);
   IF #_w2 THEN RESET_TIMER(#"TIMER 1"); END_IF;
   #"COUNTER1 2".CTU(CU := #_w1 AND #"COUNTER1 1".QU,
                     R := #RESET,
                     PV := #"SET TIME",
                     CV => #"PRESENT VALUE OF TIME");
   #BIT := #"COUNTER1 1".QU;
   #DONE := #"COUNTER1 2".QU;
END_REGION
END_FUNCTION_BLOCK

FUNCTION "mfg filtration LOGIC" : Void   // FC8, LAD
{ S7_Optimized_Access := 'TRUE' }
// stored: SetENOAutomatically false
   VAR_TEMP   // added for the SCL form of the ladder/FBD networks
      _w1 : Bool;
   END_VAR
BEGIN

REGION Network 1: MFG PROCESS START
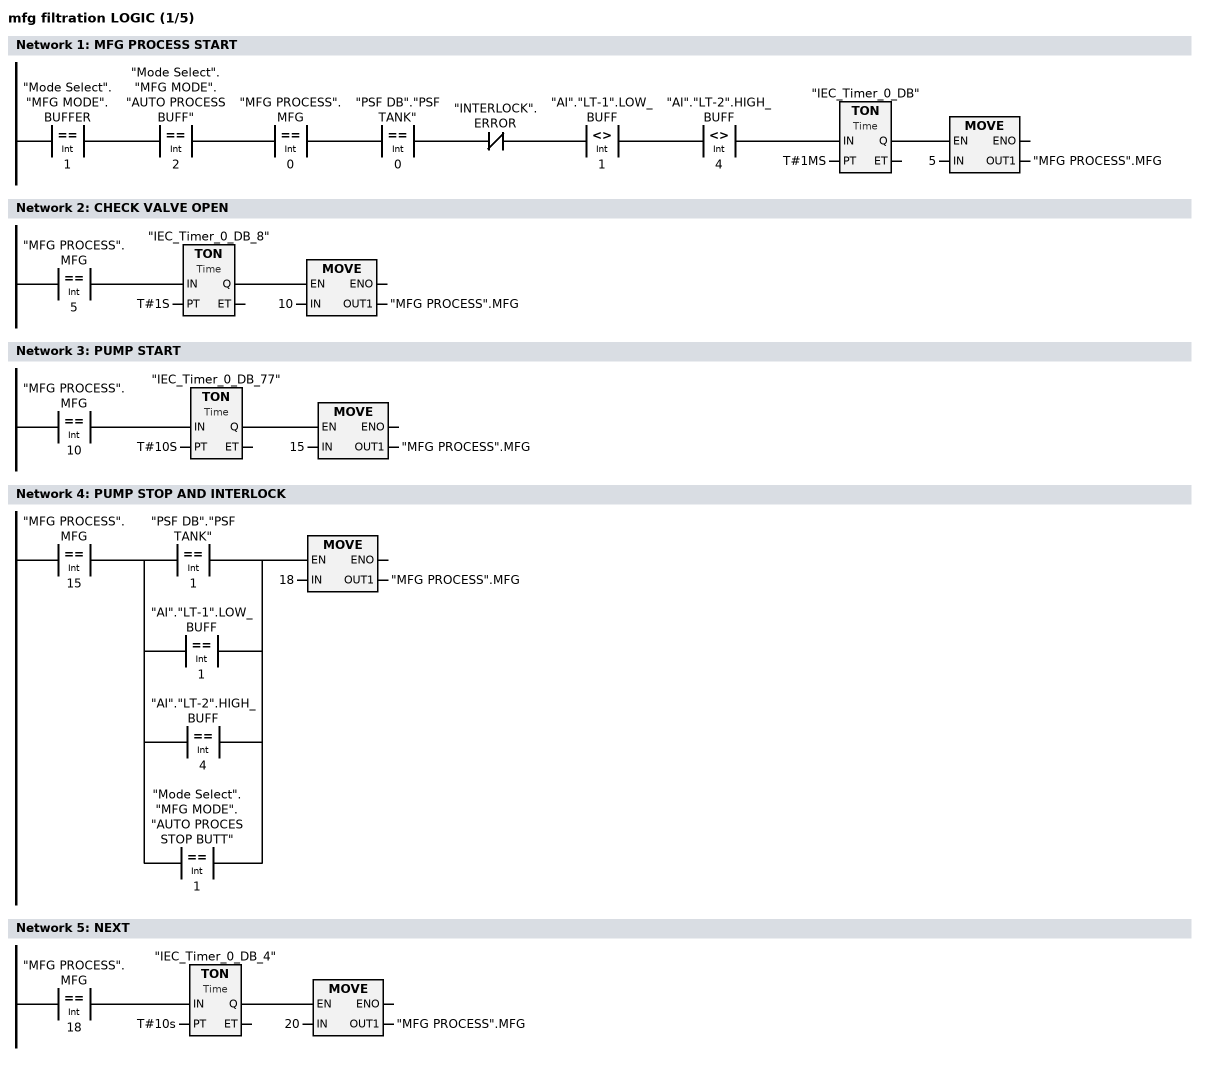
   RUNG wire#powerrail
      { S7_Templates := "SrcType := Int" } EQ_Contact(in1 := "Mode Select"."MFG MODE".BUFFER, in2 := 1)
      { S7_Templates := "SrcType := Int" } EQ_Contact(in1 := "Mode Select"."MFG MODE"."AUTO PROCESS BUFF", in2 := 2)
      { S7_Templates := "SrcType := Int" } EQ_Contact(in1 := "MFG PROCESS".MFG, in2 := 0)
      { S7_Templates := "SrcType := Int" } EQ_Contact(in1 := "PSF DB"."PSF TANK", in2 := 0)
      I_Contact( "INTERLOCK".ERROR )
      { S7_Templates := "SrcType := Int" } NE_Contact(in1 := "AI"."LT-1".LOW_BUFF, in2 := 1)
      { S7_Templates := "SrcType := Int" } NE_Contact(in1 := "AI"."LT-2".HIGH_BUFF, in2 := 4)
      { S7_Templates := "time_type := Time" } "IEC_Timer_0_DB".TON(pt := T#1MS, et =>)
      Move(in := 5, out1 => "MFG PROCESS".MFG)
   END_RUNG
   // the same network as SCL:
   "IEC_Timer_0_DB".TON(IN := ("Mode Select"."MFG MODE".BUFFER = 1) AND ("Mode Select"."MFG MODE"."AUTO PROCESS BUFF" = 2) AND ("MFG PROCESS".MFG = 0) AND ("PSF DB"."PSF TANK" = 0) AND NOT "INTERLOCK".ERROR AND ("AI"."LT-1".LOW_BUFF <> 1) AND ("AI"."LT-2".HIGH_BUFF <> 4),
                        PT := T#1MS);
   IF "IEC_Timer_0_DB".Q THEN "MFG PROCESS".MFG := 5; END_IF;
END_REGION

REGION Network 2: CHECK VALVE OPEN
   RUNG wire#powerrail
      { S7_Templates := "SrcType := Int" } EQ_Contact(in1 := "MFG PROCESS".MFG, in2 := 5)
      { S7_Templates := "time_type := Time" } "IEC_Timer_0_DB_8".TON(pt := T#1S, et =>)
      Move(in := 10, out1 => "MFG PROCESS".MFG)
   END_RUNG
   // the same network as SCL:
   "IEC_Timer_0_DB_8".TON(IN := "MFG PROCESS".MFG = 5, PT := T#1S);
   IF "IEC_Timer_0_DB_8".Q THEN "MFG PROCESS".MFG := 10; END_IF;
END_REGION

REGION Network 3: PUMP START
   RUNG wire#powerrail
      { S7_Templates := "SrcType := Int" } EQ_Contact(in1 := "MFG PROCESS".MFG, in2 := 10)
      { S7_Templates := "time_type := Time" } "IEC_Timer_0_DB_77".TON(pt := T#10S, et =>)
      Move(in := 15, out1 => "MFG PROCESS".MFG)
   END_RUNG
   // the same network as SCL:
   "IEC_Timer_0_DB_77".TON(IN := "MFG PROCESS".MFG = 10, PT := T#10S);
   IF "IEC_Timer_0_DB_77".Q THEN "MFG PROCESS".MFG := 15; END_IF;
END_REGION

REGION Network 4: PUMP STOP AND INTERLOCK
   RUNG wire#powerrail
      { S7_Templates := "SrcType := Int" } EQ_Contact(in1 := "MFG PROCESS".MFG, in2 := 15)
      wire#w1
      { S7_Templates := "SrcType := Int" } EQ_Contact(in1 := "PSF DB"."PSF TANK", in2 := 1)
      wire#w2
      Move(in := 18, out1 => "MFG PROCESS".MFG)
   END_RUNG
   RUNG wire#w1
      { S7_Templates := "SrcType := Int" } EQ_Contact(in1 := "AI"."LT-1".LOW_BUFF, in2 := 1)
   END_RUNG wire#w2
   RUNG wire#w1
      { S7_Templates := "SrcType := Int" } EQ_Contact(in1 := "AI"."LT-2".HIGH_BUFF, in2 := 4)
   END_RUNG wire#w2
   RUNG wire#w1
      { S7_Templates := "SrcType := Int" } EQ_Contact(in1 := "Mode Select"."MFG MODE"."AUTO PROCES STOP BUTT", in2 := 1)
   END_RUNG wire#w2
   // the same network as SCL:
   IF ("MFG PROCESS".MFG = 15) AND (("PSF DB"."PSF TANK" = 1) OR ("AI"."LT-1".LOW_BUFF = 1) OR ("AI"."LT-2".HIGH_BUFF = 4) OR ("Mode Select"."MFG MODE"."AUTO PROCES STOP BUTT" = 1)) THEN
       "MFG PROCESS".MFG := 18;
   END_IF;
END_REGION

REGION Network 5: NEXT
   RUNG wire#powerrail
      { S7_Templates := "SrcType := Int" } EQ_Contact(in1 := "MFG PROCESS".MFG, in2 := 18)
      { S7_Templates := "time_type := Time" } "IEC_Timer_0_DB_4".TON(pt := T#10s, et =>)
      Move(in := 20, out1 => "MFG PROCESS".MFG)
   END_RUNG
   // the same network as SCL:
   "IEC_Timer_0_DB_4".TON(IN := "MFG PROCESS".MFG = 18, PT := T#10s);
   IF "IEC_Timer_0_DB_4".Q THEN "MFG PROCESS".MFG := 20; END_IF;
END_REGION

REGION Network 6: MFG PROCESS OVER
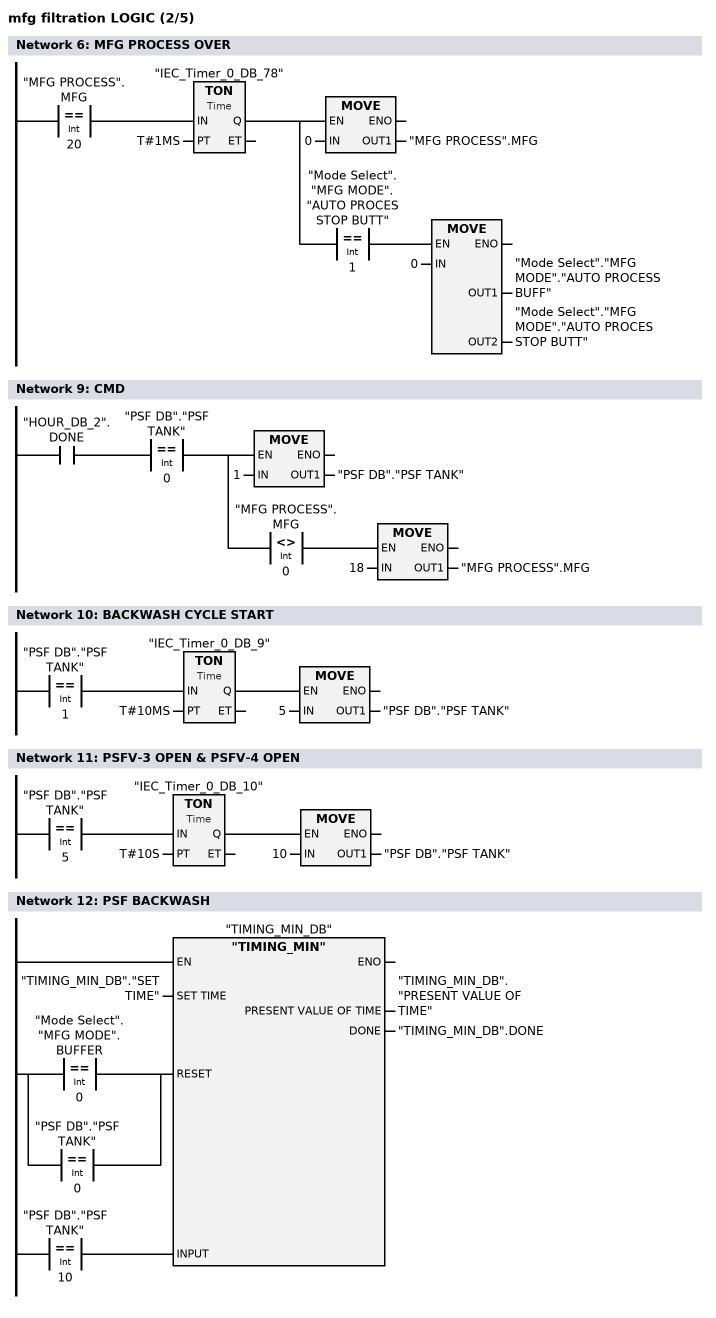
   RUNG wire#powerrail
      { S7_Templates := "SrcType := Int" } EQ_Contact(in1 := "MFG PROCESS".MFG, in2 := 20)
      { S7_Templates := "time_type := Time" } "IEC_Timer_0_DB_78".TON(pt := T#1MS, et =>)
      wire#w1
      Move(in := 0, out1 => "MFG PROCESS".MFG)
   END_RUNG
   RUNG wire#w1
      { S7_Templates := "SrcType := Int" } EQ_Contact(in1 := "Mode Select"."MFG MODE"."AUTO PROCES STOP BUTT", in2 := 1)
      Move(in := 0, out1 => "Mode Select"."MFG MODE"."AUTO PROCESS BUFF", out2 => "Mode Select"."MFG MODE"."AUTO PROCES STOP BUTT")
   END_RUNG
   // the same network as SCL:
   "IEC_Timer_0_DB_78".TON(IN := "MFG PROCESS".MFG = 20, PT := T#1MS);
   IF "IEC_Timer_0_DB_78".Q THEN "MFG PROCESS".MFG := 0; END_IF;
   IF "IEC_Timer_0_DB_78".Q AND ("Mode Select"."MFG MODE"."AUTO PROCES STOP BUTT" = 1) THEN
       "Mode Select"."MFG MODE"."AUTO PROCESS BUFF" := 0;
       "Mode Select"."MFG MODE"."AUTO PROCES STOP BUTT" := 0;
   END_IF;
END_REGION

REGION Network 9: CMD
   RUNG wire#powerrail
      Contact( "HOUR_DB_2".DONE )
      { S7_Templates := "SrcType := Int" } EQ_Contact(in1 := "PSF DB"."PSF TANK", in2 := 0)
      wire#w1
      Move(in := 1, out1 => "PSF DB"."PSF TANK")
   END_RUNG
   RUNG wire#w1
      { S7_Templates := "SrcType := Int" } NE_Contact(in1 := "MFG PROCESS".MFG, in2 := 0)
      Move(in := 18, out1 => "MFG PROCESS".MFG)
   END_RUNG
   // the same network as SCL:
   #_w1 := "HOUR_DB_2".DONE AND ("PSF DB"."PSF TANK" = 0);
   IF #_w1 THEN "PSF DB"."PSF TANK" := 1; END_IF;
   IF #_w1 AND ("MFG PROCESS".MFG <> 0) THEN "MFG PROCESS".MFG := 18; END_IF;
END_REGION

REGION Network 10: BACKWASH CYCLE START
   RUNG wire#powerrail
      { S7_Templates := "SrcType := Int" } EQ_Contact(in1 := "PSF DB"."PSF TANK", in2 := 1)
      { S7_Templates := "time_type := Time" } "IEC_Timer_0_DB_9".TON(pt := T#10MS, et =>)
      Move(in := 5, out1 => "PSF DB"."PSF TANK")
   END_RUNG
   // the same network as SCL:
   "IEC_Timer_0_DB_9".TON(IN := "PSF DB"."PSF TANK" = 1, PT := T#10MS);
   IF "IEC_Timer_0_DB_9".Q THEN "PSF DB"."PSF TANK" := 5; END_IF;
END_REGION

REGION Network 11: PSFV-3 OPEN & PSFV-4 OPEN
   RUNG wire#powerrail
      { S7_Templates := "SrcType := Int" } EQ_Contact(in1 := "PSF DB"."PSF TANK", in2 := 5)
      { S7_Templates := "time_type := Time" } "IEC_Timer_0_DB_10".TON(pt := T#10S, et =>)
      Move(in := 10, out1 => "PSF DB"."PSF TANK")
   END_RUNG
   // the same network as SCL:
   "IEC_Timer_0_DB_10".TON(IN := "PSF DB"."PSF TANK" = 5, PT := T#10S);
   IF "IEC_Timer_0_DB_10".Q THEN "PSF DB"."PSF TANK" := 10; END_IF;
END_REGION

REGION Network 12: PSF BACKWASH
   RUNG wire#powerrail
      "TIMING_MIN_DB"(RESET := wire#w1, INPUT := wire#w2, "SET TIME" := "TIMING_MIN_DB"."SET TIME", "PRESENT VALUE OF TIME" => "TIMING_MIN_DB"."PRESENT VALUE OF TIME", DONE => "TIMING_MIN_DB".DONE)
   END_RUNG
   RUNG wire#powerrail
      { S7_Templates := "SrcType := Int" } EQ_Contact(in1 := "Mode Select"."MFG MODE".BUFFER, in2 := 0)
   END_RUNG wire#w1
   RUNG wire#powerrail
      { S7_Templates := "SrcType := Int" } EQ_Contact(in1 := "PSF DB"."PSF TANK", in2 := 0)
   END_RUNG wire#w1
   RUNG wire#powerrail
      { S7_Templates := "SrcType := Int" } EQ_Contact(in1 := "PSF DB"."PSF TANK", in2 := 10)
   END_RUNG wire#w2
   // the same network as SCL:
   "TIMING_MIN_DB"("SET TIME" := "TIMING_MIN_DB"."SET TIME",   // "TIMING_MIN"
                   RESET := ("Mode Select"."MFG MODE".BUFFER = 0) OR ("PSF DB"."PSF TANK" = 0),
                   INPUT := "PSF DB"."PSF TANK" = 10,
                   "PRESENT VALUE OF TIME" => "TIMING_MIN_DB"."PRESENT VALUE OF TIME",
                   DONE => "TIMING_MIN_DB".DONE);
END_REGION

REGION Network 13: TIMER DONE
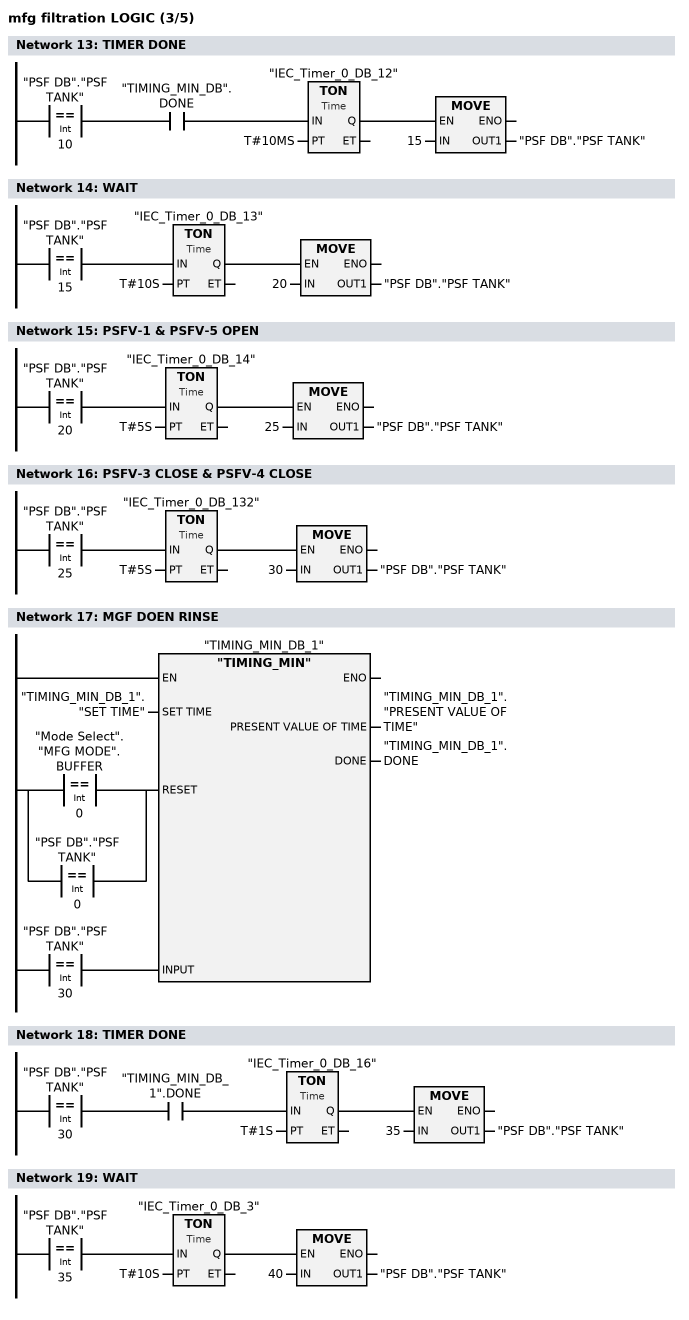
   RUNG wire#powerrail
      { S7_Templates := "SrcType := Int" } EQ_Contact(in1 := "PSF DB"."PSF TANK", in2 := 10)
      Contact( "TIMING_MIN_DB".DONE )
      { S7_Templates := "time_type := Time" } "IEC_Timer_0_DB_12".TON(pt := T#10MS, et =>)
      Move(in := 15, out1 => "PSF DB"."PSF TANK")
   END_RUNG
   // the same network as SCL:
   "IEC_Timer_0_DB_12".TON(IN := ("PSF DB"."PSF TANK" = 10) AND "TIMING_MIN_DB".DONE, PT := T#10MS);
   IF "IEC_Timer_0_DB_12".Q THEN "PSF DB"."PSF TANK" := 15; END_IF;
END_REGION

REGION Network 14: WAIT
   RUNG wire#powerrail
      { S7_Templates := "SrcType := Int" } EQ_Contact(in1 := "PSF DB"."PSF TANK", in2 := 15)
      { S7_Templates := "time_type := Time" } "IEC_Timer_0_DB_13".TON(pt := T#10S, et =>)
      Move(in := 20, out1 => "PSF DB"."PSF TANK")
   END_RUNG
   // the same network as SCL:
   "IEC_Timer_0_DB_13".TON(IN := "PSF DB"."PSF TANK" = 15, PT := T#10S);
   IF "IEC_Timer_0_DB_13".Q THEN "PSF DB"."PSF TANK" := 20; END_IF;
END_REGION

REGION Network 15: PSFV-1 & PSFV-5 OPEN
   RUNG wire#powerrail
      { S7_Templates := "SrcType := Int" } EQ_Contact(in1 := "PSF DB"."PSF TANK", in2 := 20)
      { S7_Templates := "time_type := Time" } "IEC_Timer_0_DB_14".TON(pt := T#5S, et =>)
      Move(in := 25, out1 => "PSF DB"."PSF TANK")
   END_RUNG
   // the same network as SCL:
   "IEC_Timer_0_DB_14".TON(IN := "PSF DB"."PSF TANK" = 20, PT := T#5S);
   IF "IEC_Timer_0_DB_14".Q THEN "PSF DB"."PSF TANK" := 25; END_IF;
END_REGION

REGION Network 16: PSFV-3 CLOSE & PSFV-4 CLOSE
   RUNG wire#powerrail
      { S7_Templates := "SrcType := Int" } EQ_Contact(in1 := "PSF DB"."PSF TANK", in2 := 25)
      { S7_Templates := "time_type := Time" } "IEC_Timer_0_DB_132".TON(pt := T#5S, et =>)
      Move(in := 30, out1 => "PSF DB"."PSF TANK")
   END_RUNG
   // the same network as SCL:
   "IEC_Timer_0_DB_132".TON(IN := "PSF DB"."PSF TANK" = 25, PT := T#5S);
   IF "IEC_Timer_0_DB_132".Q THEN "PSF DB"."PSF TANK" := 30; END_IF;
END_REGION

REGION Network 17: MGF DOEN RINSE
   RUNG wire#powerrail
      "TIMING_MIN_DB_1"(RESET := wire#w1, INPUT := wire#w2, "SET TIME" := "TIMING_MIN_DB_1"."SET TIME", "PRESENT VALUE OF TIME" => "TIMING_MIN_DB_1"."PRESENT VALUE OF TIME", DONE => "TIMING_MIN_DB_1".DONE)
   END_RUNG
   RUNG wire#powerrail
      { S7_Templates := "SrcType := Int" } EQ_Contact(in1 := "Mode Select"."MFG MODE".BUFFER, in2 := 0)
   END_RUNG wire#w1
   RUNG wire#powerrail
      { S7_Templates := "SrcType := Int" } EQ_Contact(in1 := "PSF DB"."PSF TANK", in2 := 0)
   END_RUNG wire#w1
   RUNG wire#powerrail
      { S7_Templates := "SrcType := Int" } EQ_Contact(in1 := "PSF DB"."PSF TANK", in2 := 30)
   END_RUNG wire#w2
   // the same network as SCL:
   "TIMING_MIN_DB_1"("SET TIME" := "TIMING_MIN_DB_1"."SET TIME",   // "TIMING_MIN"
                     RESET := ("Mode Select"."MFG MODE".BUFFER = 0) OR ("PSF DB"."PSF TANK" = 0),
                     INPUT := "PSF DB"."PSF TANK" = 30,
                     "PRESENT VALUE OF TIME" => "TIMING_MIN_DB_1"."PRESENT VALUE OF TIME",
                     DONE => "TIMING_MIN_DB_1".DONE);
END_REGION

REGION Network 18: TIMER DONE
   RUNG wire#powerrail
      { S7_Templates := "SrcType := Int" } EQ_Contact(in1 := "PSF DB"."PSF TANK", in2 := 30)
      Contact( "TIMING_MIN_DB_1".DONE )
      { S7_Templates := "time_type := Time" } "IEC_Timer_0_DB_16".TON(pt := T#1S, et =>)
      Move(in := 35, out1 => "PSF DB"."PSF TANK")
   END_RUNG
   // the same network as SCL:
   "IEC_Timer_0_DB_16".TON(IN := ("PSF DB"."PSF TANK" = 30) AND "TIMING_MIN_DB_1".DONE, PT := T#1S);
   IF "IEC_Timer_0_DB_16".Q THEN "PSF DB"."PSF TANK" := 35; END_IF;
END_REGION

REGION Network 19: WAIT
   RUNG wire#powerrail
      { S7_Templates := "SrcType := Int" } EQ_Contact(in1 := "PSF DB"."PSF TANK", in2 := 35)
      { S7_Templates := "time_type := Time" } "IEC_Timer_0_DB_3".TON(pt := T#10S, et =>)
      Move(in := 40, out1 => "PSF DB"."PSF TANK")
   END_RUNG
   // the same network as SCL:
   "IEC_Timer_0_DB_3".TON(IN := "PSF DB"."PSF TANK" = 35, PT := T#10S);
   IF "IEC_Timer_0_DB_3".Q THEN "PSF DB"."PSF TANK" := 40; END_IF;
END_REGION

REGION Network 20: PSFV1 & PSFV2 & ACFV3 & ACFV4 OPEN
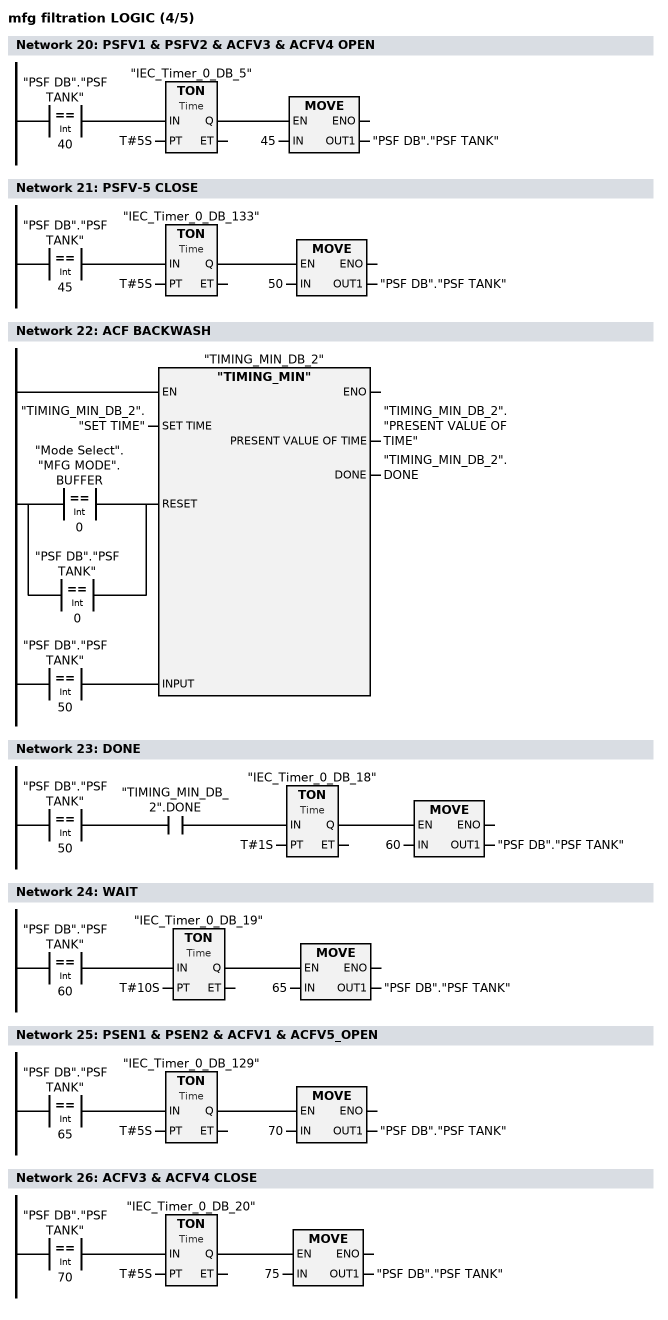
   RUNG wire#powerrail
      { S7_Templates := "SrcType := Int" } EQ_Contact(in1 := "PSF DB"."PSF TANK", in2 := 40)
      { S7_Templates := "time_type := Time" } "IEC_Timer_0_DB_5".TON(pt := T#5S, et =>)
      Move(in := 45, out1 => "PSF DB"."PSF TANK")
   END_RUNG
   // the same network as SCL:
   "IEC_Timer_0_DB_5".TON(IN := "PSF DB"."PSF TANK" = 40, PT := T#5S);
   IF "IEC_Timer_0_DB_5".Q THEN "PSF DB"."PSF TANK" := 45; END_IF;
END_REGION

REGION Network 21: PSFV-5 CLOSE
   RUNG wire#powerrail
      { S7_Templates := "SrcType := Int" } EQ_Contact(in1 := "PSF DB"."PSF TANK", in2 := 45)
      { S7_Templates := "time_type := Time" } "IEC_Timer_0_DB_133".TON(pt := T#5S, et =>)
      Move(in := 50, out1 => "PSF DB"."PSF TANK")
   END_RUNG
   // the same network as SCL:
   "IEC_Timer_0_DB_133".TON(IN := "PSF DB"."PSF TANK" = 45, PT := T#5S);
   IF "IEC_Timer_0_DB_133".Q THEN "PSF DB"."PSF TANK" := 50; END_IF;
END_REGION

REGION Network 22: ACF BACKWASH
   RUNG wire#powerrail
      "TIMING_MIN_DB_2"(RESET := wire#w1, INPUT := wire#w2, "SET TIME" := "TIMING_MIN_DB_2"."SET TIME", "PRESENT VALUE OF TIME" => "TIMING_MIN_DB_2"."PRESENT VALUE OF TIME", DONE => "TIMING_MIN_DB_2".DONE)
   END_RUNG
   RUNG wire#powerrail
      { S7_Templates := "SrcType := Int" } EQ_Contact(in1 := "Mode Select"."MFG MODE".BUFFER, in2 := 0)
   END_RUNG wire#w1
   RUNG wire#powerrail
      { S7_Templates := "SrcType := Int" } EQ_Contact(in1 := "PSF DB"."PSF TANK", in2 := 0)
   END_RUNG wire#w1
   RUNG wire#powerrail
      { S7_Templates := "SrcType := Int" } EQ_Contact(in1 := "PSF DB"."PSF TANK", in2 := 50)
   END_RUNG wire#w2
   // the same network as SCL:
   "TIMING_MIN_DB_2"("SET TIME" := "TIMING_MIN_DB_2"."SET TIME",   // "TIMING_MIN"
                     RESET := ("Mode Select"."MFG MODE".BUFFER = 0) OR ("PSF DB"."PSF TANK" = 0),
                     INPUT := "PSF DB"."PSF TANK" = 50,
                     "PRESENT VALUE OF TIME" => "TIMING_MIN_DB_2"."PRESENT VALUE OF TIME",
                     DONE => "TIMING_MIN_DB_2".DONE);
END_REGION

REGION Network 23: DONE
   RUNG wire#powerrail
      { S7_Templates := "SrcType := Int" } EQ_Contact(in1 := "PSF DB"."PSF TANK", in2 := 50)
      Contact( "TIMING_MIN_DB_2".DONE )
      { S7_Templates := "time_type := Time" } "IEC_Timer_0_DB_18".TON(pt := T#1S, et =>)
      Move(in := 60, out1 => "PSF DB"."PSF TANK")
   END_RUNG
   // the same network as SCL:
   "IEC_Timer_0_DB_18".TON(IN := ("PSF DB"."PSF TANK" = 50) AND "TIMING_MIN_DB_2".DONE, PT := T#1S);
   IF "IEC_Timer_0_DB_18".Q THEN "PSF DB"."PSF TANK" := 60; END_IF;
END_REGION

REGION Network 24: WAIT
   RUNG wire#powerrail
      { S7_Templates := "SrcType := Int" } EQ_Contact(in1 := "PSF DB"."PSF TANK", in2 := 60)
      { S7_Templates := "time_type := Time" } "IEC_Timer_0_DB_19".TON(pt := T#10S, et =>)
      Move(in := 65, out1 => "PSF DB"."PSF TANK")
   END_RUNG
   // the same network as SCL:
   "IEC_Timer_0_DB_19".TON(IN := "PSF DB"."PSF TANK" = 60, PT := T#10S);
   IF "IEC_Timer_0_DB_19".Q THEN "PSF DB"."PSF TANK" := 65; END_IF;
END_REGION

REGION Network 25: PSEN1 & PSEN2 & ACFV1 & ACFV5_OPEN
   RUNG wire#powerrail
      { S7_Templates := "SrcType := Int" } EQ_Contact(in1 := "PSF DB"."PSF TANK", in2 := 65)
      { S7_Templates := "time_type := Time" } "IEC_Timer_0_DB_129".TON(pt := T#5S, et =>)
      Move(in := 70, out1 => "PSF DB"."PSF TANK")
   END_RUNG
   // the same network as SCL:
   "IEC_Timer_0_DB_129".TON(IN := "PSF DB"."PSF TANK" = 65, PT := T#5S);
   IF "IEC_Timer_0_DB_129".Q THEN "PSF DB"."PSF TANK" := 70; END_IF;
END_REGION

REGION Network 26: ACFV3 & ACFV4 CLOSE
   RUNG wire#powerrail
      { S7_Templates := "SrcType := Int" } EQ_Contact(in1 := "PSF DB"."PSF TANK", in2 := 70)
      { S7_Templates := "time_type := Time" } "IEC_Timer_0_DB_20".TON(pt := T#5S, et =>)
      Move(in := 75, out1 => "PSF DB"."PSF TANK")
   END_RUNG
   // the same network as SCL:
   "IEC_Timer_0_DB_20".TON(IN := "PSF DB"."PSF TANK" = 70, PT := T#5S);
   IF "IEC_Timer_0_DB_20".Q THEN "PSF DB"."PSF TANK" := 75; END_IF;
END_REGION

REGION Network 27: ACF DOWN RINSE
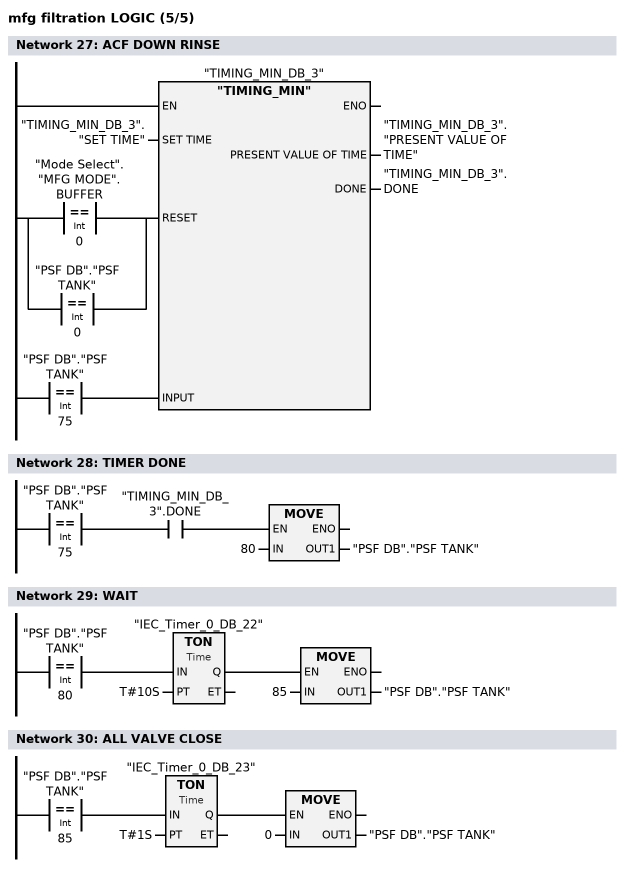
   RUNG wire#powerrail
      "TIMING_MIN_DB_3"(RESET := wire#w1, INPUT := wire#w2, "SET TIME" := "TIMING_MIN_DB_3"."SET TIME", "PRESENT VALUE OF TIME" => "TIMING_MIN_DB_3"."PRESENT VALUE OF TIME", DONE => "TIMING_MIN_DB_3".DONE)
   END_RUNG
   RUNG wire#powerrail
      { S7_Templates := "SrcType := Int" } EQ_Contact(in1 := "Mode Select"."MFG MODE".BUFFER, in2 := 0)
   END_RUNG wire#w1
   RUNG wire#powerrail
      { S7_Templates := "SrcType := Int" } EQ_Contact(in1 := "PSF DB"."PSF TANK", in2 := 0)
   END_RUNG wire#w1
   RUNG wire#powerrail
      { S7_Templates := "SrcType := Int" } EQ_Contact(in1 := "PSF DB"."PSF TANK", in2 := 75)
   END_RUNG wire#w2
   // the same network as SCL:
   "TIMING_MIN_DB_3"("SET TIME" := "TIMING_MIN_DB_3"."SET TIME",   // "TIMING_MIN"
                     RESET := ("Mode Select"."MFG MODE".BUFFER = 0) OR ("PSF DB"."PSF TANK" = 0),
                     INPUT := "PSF DB"."PSF TANK" = 75,
                     "PRESENT VALUE OF TIME" => "TIMING_MIN_DB_3"."PRESENT VALUE OF TIME",
                     DONE => "TIMING_MIN_DB_3".DONE);
END_REGION

REGION Network 28: TIMER DONE
   RUNG wire#powerrail
      { S7_Templates := "SrcType := Int" } EQ_Contact(in1 := "PSF DB"."PSF TANK", in2 := 75)
      Contact( "TIMING_MIN_DB_3".DONE )
      Move(in := 80, out1 => "PSF DB"."PSF TANK")
   END_RUNG
   // the same network as SCL:
   IF ("PSF DB"."PSF TANK" = 75) AND "TIMING_MIN_DB_3".DONE THEN "PSF DB"."PSF TANK" := 80; END_IF;
END_REGION

REGION Network 29: WAIT
   RUNG wire#powerrail
      { S7_Templates := "SrcType := Int" } EQ_Contact(in1 := "PSF DB"."PSF TANK", in2 := 80)
      { S7_Templates := "time_type := Time" } "IEC_Timer_0_DB_22".TON(pt := T#10S, et =>)
      Move(in := 85, out1 => "PSF DB"."PSF TANK")
   END_RUNG
   // the same network as SCL:
   "IEC_Timer_0_DB_22".TON(IN := "PSF DB"."PSF TANK" = 80, PT := T#10S);
   IF "IEC_Timer_0_DB_22".Q THEN "PSF DB"."PSF TANK" := 85; END_IF;
END_REGION

REGION Network 30: ALL VALVE CLOSE
   RUNG wire#powerrail
      { S7_Templates := "SrcType := Int" } EQ_Contact(in1 := "PSF DB"."PSF TANK", in2 := 85)
      { S7_Templates := "time_type := Time" } "IEC_Timer_0_DB_23".TON(pt := T#1S, et =>)
      Move(in := 0, out1 => "PSF DB"."PSF TANK")
   END_RUNG
   // the same network as SCL:
   "IEC_Timer_0_DB_23".TON(IN := "PSF DB"."PSF TANK" = 85, PT := T#1S);
   IF "IEC_Timer_0_DB_23".Q THEN "PSF DB"."PSF TANK" := 0; END_IF;
END_REGION
END_FUNCTION

FUNCTION_BLOCK "TIMING_MIN"   // FB3, LAD
{ S7_Optimized_Access := 'TRUE' }
// stored: MemoryReserve 100, SetENOAutomatically false
   VAR_INPUT
      "SET TIME" : Int;
      RESET : Bool;
      INPUT : Bool;
   END_VAR
   VAR_OUTPUT
      "PRESENT VALUE OF TIME" : Int;
      DONE : Bool;
   END_VAR
   VAR
      "TIMER 1" { S7_SetPoint := 'True'} : IEC_TIMER;
   END_VAR
   VAR RETAIN
      "COUNTER1 1" { S7_SetPoint := 'True'} : IEC_COUNTER;
   END_VAR
   VAR_TEMP   // added for the SCL form of the ladder/FBD networks
      _w1 : Bool;
      _w2 : Bool;
   END_VAR
BEGIN

REGION Network 1
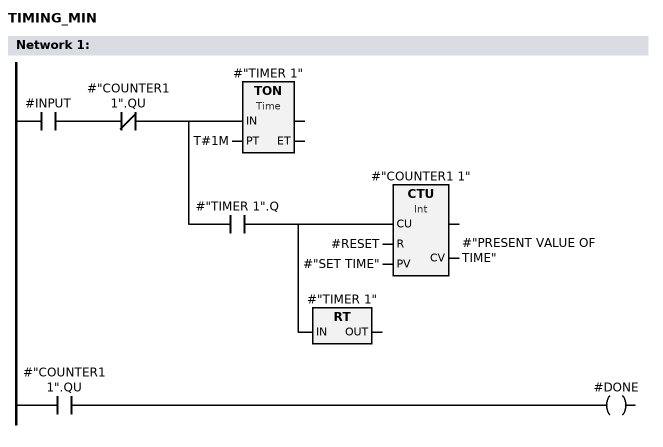
   RUNG wire#powerrail
      Contact( #INPUT )
      I_Contact( #"COUNTER1 1".QU )
      wire#w1
      { S7_Templates := "time_type := Time" } #"TIMER 1".TON(pt := T#1M, et =>)
   END_RUNG
   RUNG wire#w1
      Contact( #"TIMER 1".Q )
      wire#w2
      { S7_Templates := "value_type := Int" } #"COUNTER1 1".CTU(r := #RESET, pv := #"SET TIME", cv => #"PRESENT VALUE OF TIME")
   END_RUNG
   RUNG wire#w2
      RT_Coil( #"TIMER 1" )
   END_RUNG
   RUNG wire#powerrail
      Contact( #"COUNTER1 1".QU )
      Coil( #DONE )
   END_RUNG
   // the same network as SCL:
   #_w1 := #INPUT AND NOT #"COUNTER1 1".QU;
   #"TIMER 1".TON(IN := #_w1, PT := T#1M);
   #_w2 := #_w1 AND #"TIMER 1".Q;
   #"COUNTER1 1".CTU(CU := #_w2, R := #RESET, PV := #"SET TIME", CV => #"PRESENT VALUE OF TIME");
   IF #_w2 THEN RESET_TIMER(#"TIMER 1"); END_IF;
   #DONE := #"COUNTER1 1".QU;
END_REGION
END_FUNCTION_BLOCK

FUNCTION "MFG OUTPUT SECTION" : Void   // FC10, LAD
{ S7_Optimized_Access := 'TRUE' }
// stored: SetENOAutomatically false
   VAR_TEMP   // added for the SCL form of the ladder/FBD networks
      _w1 : Bool;
   END_VAR
BEGIN

REGION Network 1: PSFV-1 – OPEN
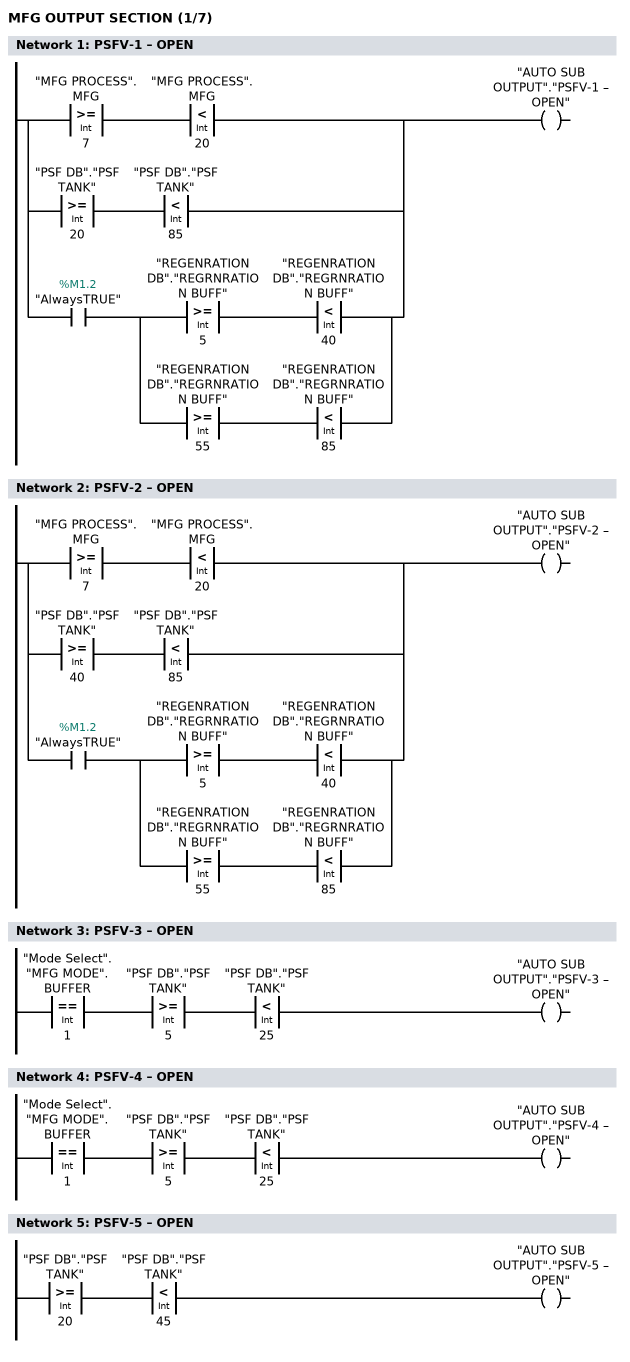
   RUNG wire#powerrail
      { S7_Templates := "SrcType := Int" } GE_Contact(in1 := "MFG PROCESS".MFG, in2 := 7)
      { S7_Templates := "SrcType := Int" } LT_Contact(in1 := "MFG PROCESS".MFG, in2 := 20)
      wire#w1
      Coil( "AUTO SUB OUTPUT"."PSFV-1 – OPEN" )
   END_RUNG
   RUNG wire#powerrail
      { S7_Templates := "SrcType := Int" } GE_Contact(in1 := "PSF DB"."PSF TANK", in2 := 20)
      { S7_Templates := "SrcType := Int" } LT_Contact(in1 := "PSF DB"."PSF TANK", in2 := 85)
   END_RUNG wire#w1
   RUNG wire#powerrail
      Contact( "AlwaysTRUE" )
      wire#w2
      { S7_Templates := "SrcType := Int" } GE_Contact(in1 := "REGENRATION DB"."REGRNRATION BUFF", in2 := 5)
      { S7_Templates := "SrcType := Int" } LT_Contact(in1 := "REGENRATION DB"."REGRNRATION BUFF", in2 := 40)
   END_RUNG wire#w1
   RUNG wire#w2
      { S7_Templates := "SrcType := Int" } GE_Contact(in1 := "REGENRATION DB"."REGRNRATION BUFF", in2 := 55)
      { S7_Templates := "SrcType := Int" } LT_Contact(in1 := "REGENRATION DB"."REGRNRATION BUFF", in2 := 85)
   END_RUNG wire#w1
   // the same network as SCL:
   "AUTO SUB OUTPUT"."PSFV-1 – OPEN" := (("MFG PROCESS".MFG >= 7) AND ("MFG PROCESS".MFG < 20)) OR (("PSF DB"."PSF TANK" >= 20) AND ("PSF DB"."PSF TANK" < 85)) OR ("AlwaysTRUE" AND ((("REGENRATION DB"."REGRNRATION BUFF" >= 5) AND ("REGENRATION DB"."REGRNRATION BUFF" < 40)) OR (("REGENRATION DB"."REGRNRATION BUFF" >= 55) AND ("REGENRATION DB"."REGRNRATION BUFF" < 85))));
END_REGION

REGION Network 2: PSFV-2 – OPEN
   RUNG wire#powerrail
      { S7_Templates := "SrcType := Int" } GE_Contact(in1 := "MFG PROCESS".MFG, in2 := 7)
      { S7_Templates := "SrcType := Int" } LT_Contact(in1 := "MFG PROCESS".MFG, in2 := 20)
      wire#w1
      Coil( "AUTO SUB OUTPUT"."PSFV-2 – OPEN" )
   END_RUNG
   RUNG wire#powerrail
      { S7_Templates := "SrcType := Int" } GE_Contact(in1 := "PSF DB"."PSF TANK", in2 := 40)
      { S7_Templates := "SrcType := Int" } LT_Contact(in1 := "PSF DB"."PSF TANK", in2 := 85)
   END_RUNG wire#w1
   RUNG wire#powerrail
      Contact( "AlwaysTRUE" )
      wire#w2
      { S7_Templates := "SrcType := Int" } GE_Contact(in1 := "REGENRATION DB"."REGRNRATION BUFF", in2 := 5)
      { S7_Templates := "SrcType := Int" } LT_Contact(in1 := "REGENRATION DB"."REGRNRATION BUFF", in2 := 40)
   END_RUNG wire#w1
   RUNG wire#w2
      { S7_Templates := "SrcType := Int" } GE_Contact(in1 := "REGENRATION DB"."REGRNRATION BUFF", in2 := 55)
      { S7_Templates := "SrcType := Int" } LT_Contact(in1 := "REGENRATION DB"."REGRNRATION BUFF", in2 := 85)
   END_RUNG wire#w1
   // the same network as SCL:
   "AUTO SUB OUTPUT"."PSFV-2 – OPEN" := (("MFG PROCESS".MFG >= 7) AND ("MFG PROCESS".MFG < 20)) OR (("PSF DB"."PSF TANK" >= 40) AND ("PSF DB"."PSF TANK" < 85)) OR ("AlwaysTRUE" AND ((("REGENRATION DB"."REGRNRATION BUFF" >= 5) AND ("REGENRATION DB"."REGRNRATION BUFF" < 40)) OR (("REGENRATION DB"."REGRNRATION BUFF" >= 55) AND ("REGENRATION DB"."REGRNRATION BUFF" < 85))));
END_REGION

REGION Network 3: PSFV-3 – OPEN
   RUNG wire#powerrail
      { S7_Templates := "SrcType := Int" } EQ_Contact(in1 := "Mode Select"."MFG MODE".BUFFER, in2 := 1)
      { S7_Templates := "SrcType := Int" } GE_Contact(in1 := "PSF DB"."PSF TANK", in2 := 5)
      { S7_Templates := "SrcType := Int" } LT_Contact(in1 := "PSF DB"."PSF TANK", in2 := 25)
      Coil( "AUTO SUB OUTPUT"."PSFV-3 – OPEN" )
   END_RUNG
   // the same network as SCL:
   "AUTO SUB OUTPUT"."PSFV-3 – OPEN" := ("Mode Select"."MFG MODE".BUFFER = 1) AND ("PSF DB"."PSF TANK" >= 5) AND ("PSF DB"."PSF TANK" < 25);
END_REGION

REGION Network 4: PSFV-4 – OPEN
   RUNG wire#powerrail
      { S7_Templates := "SrcType := Int" } EQ_Contact(in1 := "Mode Select"."MFG MODE".BUFFER, in2 := 1)
      { S7_Templates := "SrcType := Int" } GE_Contact(in1 := "PSF DB"."PSF TANK", in2 := 5)
      { S7_Templates := "SrcType := Int" } LT_Contact(in1 := "PSF DB"."PSF TANK", in2 := 25)
      Coil( "AUTO SUB OUTPUT"."PSFV-4 – OPEN" )
   END_RUNG
   // the same network as SCL:
   "AUTO SUB OUTPUT"."PSFV-4 – OPEN" := ("Mode Select"."MFG MODE".BUFFER = 1) AND ("PSF DB"."PSF TANK" >= 5) AND ("PSF DB"."PSF TANK" < 25);
END_REGION

REGION Network 5: PSFV-5 – OPEN
   RUNG wire#powerrail
      { S7_Templates := "SrcType := Int" } GE_Contact(in1 := "PSF DB"."PSF TANK", in2 := 20)
      { S7_Templates := "SrcType := Int" } LT_Contact(in1 := "PSF DB"."PSF TANK", in2 := 45)
      Coil( "AUTO SUB OUTPUT"."PSFV-5 – OPEN" )
   END_RUNG
   // the same network as SCL:
   "AUTO SUB OUTPUT"."PSFV-5 – OPEN" := ("PSF DB"."PSF TANK" >= 20) AND ("PSF DB"."PSF TANK" < 45);
END_REGION

REGION Network 6: PSFV-6 – OPEN
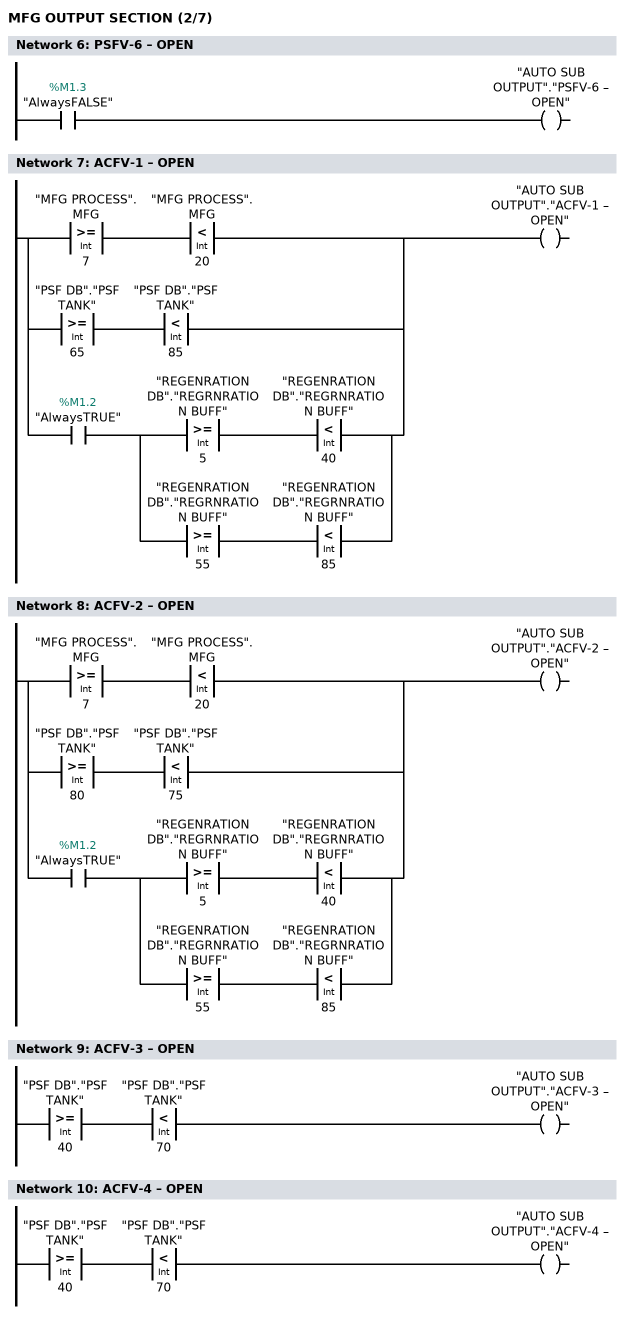
   RUNG wire#powerrail
      Contact( "AlwaysFALSE" )
      Coil( "AUTO SUB OUTPUT"."PSFV-6 – OPEN" )
   END_RUNG
   // the same network as SCL:
   "AUTO SUB OUTPUT"."PSFV-6 – OPEN" := "AlwaysFALSE";
END_REGION

REGION Network 7: ACFV-1 – OPEN
   RUNG wire#powerrail
      { S7_Templates := "SrcType := Int" } GE_Contact(in1 := "MFG PROCESS".MFG, in2 := 7)
      { S7_Templates := "SrcType := Int" } LT_Contact(in1 := "MFG PROCESS".MFG, in2 := 20)
      wire#w1
      Coil( "AUTO SUB OUTPUT"."ACFV-1 – OPEN" )
   END_RUNG
   RUNG wire#powerrail
      { S7_Templates := "SrcType := Int" } GE_Contact(in1 := "PSF DB"."PSF TANK", in2 := 65)
      { S7_Templates := "SrcType := Int" } LT_Contact(in1 := "PSF DB"."PSF TANK", in2 := 85)
   END_RUNG wire#w1
   RUNG wire#powerrail
      Contact( "AlwaysTRUE" )
      wire#w2
      { S7_Templates := "SrcType := Int" } GE_Contact(in1 := "REGENRATION DB"."REGRNRATION BUFF", in2 := 5)
      { S7_Templates := "SrcType := Int" } LT_Contact(in1 := "REGENRATION DB"."REGRNRATION BUFF", in2 := 40)
   END_RUNG wire#w1
   RUNG wire#w2
      { S7_Templates := "SrcType := Int" } GE_Contact(in1 := "REGENRATION DB"."REGRNRATION BUFF", in2 := 55)
      { S7_Templates := "SrcType := Int" } LT_Contact(in1 := "REGENRATION DB"."REGRNRATION BUFF", in2 := 85)
   END_RUNG wire#w1
   // the same network as SCL:
   "AUTO SUB OUTPUT"."ACFV-1 – OPEN" := (("MFG PROCESS".MFG >= 7) AND ("MFG PROCESS".MFG < 20)) OR (("PSF DB"."PSF TANK" >= 65) AND ("PSF DB"."PSF TANK" < 85)) OR ("AlwaysTRUE" AND ((("REGENRATION DB"."REGRNRATION BUFF" >= 5) AND ("REGENRATION DB"."REGRNRATION BUFF" < 40)) OR (("REGENRATION DB"."REGRNRATION BUFF" >= 55) AND ("REGENRATION DB"."REGRNRATION BUFF" < 85))));
END_REGION

REGION Network 8: ACFV-2 – OPEN
   RUNG wire#powerrail
      { S7_Templates := "SrcType := Int" } GE_Contact(in1 := "MFG PROCESS".MFG, in2 := 7)
      { S7_Templates := "SrcType := Int" } LT_Contact(in1 := "MFG PROCESS".MFG, in2 := 20)
      wire#w1
      Coil( "AUTO SUB OUTPUT"."ACFV-2 – OPEN" )
   END_RUNG
   RUNG wire#powerrail
      { S7_Templates := "SrcType := Int" } GE_Contact(in1 := "PSF DB"."PSF TANK", in2 := 80)
      { S7_Templates := "SrcType := Int" } LT_Contact(in1 := "PSF DB"."PSF TANK", in2 := 75)
   END_RUNG wire#w1
   RUNG wire#powerrail
      Contact( "AlwaysTRUE" )
      wire#w2
      { S7_Templates := "SrcType := Int" } GE_Contact(in1 := "REGENRATION DB"."REGRNRATION BUFF", in2 := 5)
      { S7_Templates := "SrcType := Int" } LT_Contact(in1 := "REGENRATION DB"."REGRNRATION BUFF", in2 := 40)
   END_RUNG wire#w1
   RUNG wire#w2
      { S7_Templates := "SrcType := Int" } GE_Contact(in1 := "REGENRATION DB"."REGRNRATION BUFF", in2 := 55)
      { S7_Templates := "SrcType := Int" } LT_Contact(in1 := "REGENRATION DB"."REGRNRATION BUFF", in2 := 85)
   END_RUNG wire#w1
   // the same network as SCL:
   "AUTO SUB OUTPUT"."ACFV-2 – OPEN" := (("MFG PROCESS".MFG >= 7) AND ("MFG PROCESS".MFG < 20)) OR (("PSF DB"."PSF TANK" >= 80) AND ("PSF DB"."PSF TANK" < 75)) OR ("AlwaysTRUE" AND ((("REGENRATION DB"."REGRNRATION BUFF" >= 5) AND ("REGENRATION DB"."REGRNRATION BUFF" < 40)) OR (("REGENRATION DB"."REGRNRATION BUFF" >= 55) AND ("REGENRATION DB"."REGRNRATION BUFF" < 85))));
END_REGION

REGION Network 9: ACFV-3 – OPEN
   RUNG wire#powerrail
      { S7_Templates := "SrcType := Int" } GE_Contact(in1 := "PSF DB"."PSF TANK", in2 := 40)
      { S7_Templates := "SrcType := Int" } LT_Contact(in1 := "PSF DB"."PSF TANK", in2 := 70)
      Coil( "AUTO SUB OUTPUT"."ACFV-3 – OPEN" )
   END_RUNG
   // the same network as SCL:
   "AUTO SUB OUTPUT"."ACFV-3 – OPEN" := ("PSF DB"."PSF TANK" >= 40) AND ("PSF DB"."PSF TANK" < 70);
END_REGION

REGION Network 10: ACFV-4 – OPEN
   RUNG wire#powerrail
      { S7_Templates := "SrcType := Int" } GE_Contact(in1 := "PSF DB"."PSF TANK", in2 := 40)
      { S7_Templates := "SrcType := Int" } LT_Contact(in1 := "PSF DB"."PSF TANK", in2 := 70)
      Coil( "AUTO SUB OUTPUT"."ACFV-4 – OPEN" )
   END_RUNG
   // the same network as SCL:
   "AUTO SUB OUTPUT"."ACFV-4 – OPEN" := ("PSF DB"."PSF TANK" >= 40) AND ("PSF DB"."PSF TANK" < 70);
END_REGION

REGION Network 11: ACFV-5 – OPEN
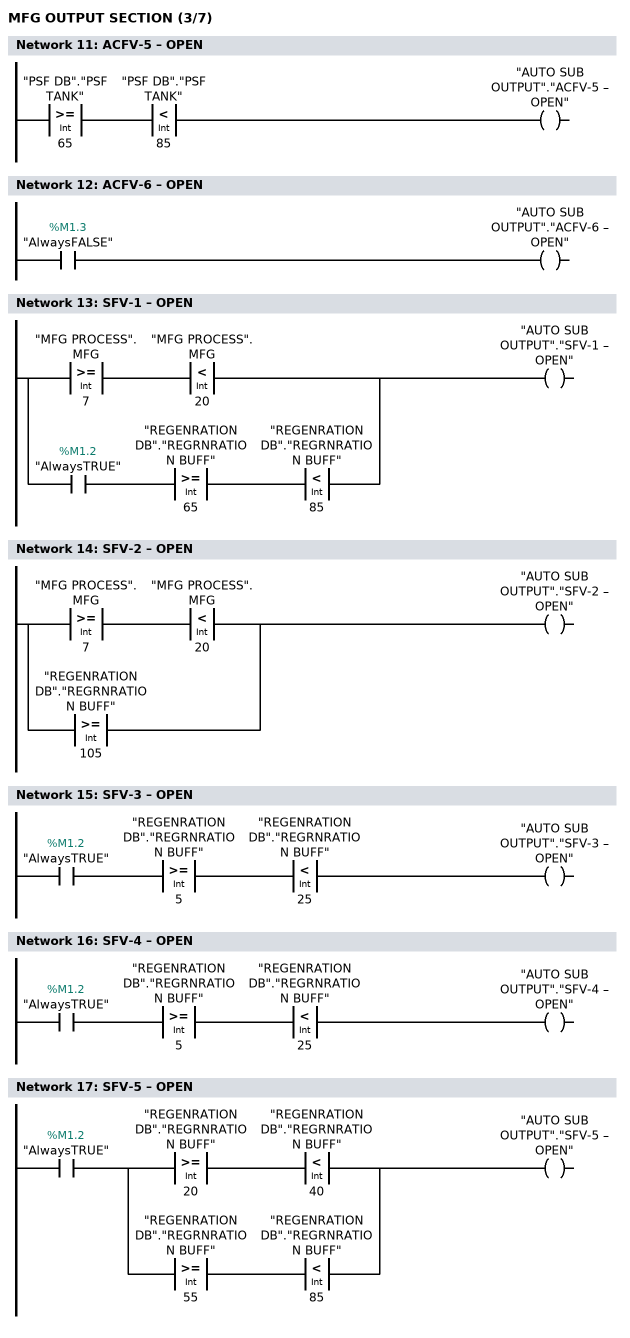
   RUNG wire#powerrail
      { S7_Templates := "SrcType := Int" } GE_Contact(in1 := "PSF DB"."PSF TANK", in2 := 65)
      { S7_Templates := "SrcType := Int" } LT_Contact(in1 := "PSF DB"."PSF TANK", in2 := 85)
      Coil( "AUTO SUB OUTPUT"."ACFV-5 – OPEN" )
   END_RUNG
   // the same network as SCL:
   "AUTO SUB OUTPUT"."ACFV-5 – OPEN" := ("PSF DB"."PSF TANK" >= 65) AND ("PSF DB"."PSF TANK" < 85);
END_REGION

REGION Network 12: ACFV-6 – OPEN
   RUNG wire#powerrail
      Contact( "AlwaysFALSE" )
      Coil( "AUTO SUB OUTPUT"."ACFV-6 – OPEN" )
   END_RUNG
   // the same network as SCL:
   "AUTO SUB OUTPUT"."ACFV-6 – OPEN" := "AlwaysFALSE";
END_REGION

REGION Network 13: SFV-1 – OPEN
   RUNG wire#powerrail
      { S7_Templates := "SrcType := Int" } GE_Contact(in1 := "MFG PROCESS".MFG, in2 := 7)
      { S7_Templates := "SrcType := Int" } LT_Contact(in1 := "MFG PROCESS".MFG, in2 := 20)
      wire#w1
      Coil( "AUTO SUB OUTPUT"."SFV-1 – OPEN" )
   END_RUNG
   RUNG wire#powerrail
      Contact( "AlwaysTRUE" )
      { S7_Templates := "SrcType := Int" } GE_Contact(in1 := "REGENRATION DB"."REGRNRATION BUFF", in2 := 65)
      { S7_Templates := "SrcType := Int" } LT_Contact(in1 := "REGENRATION DB"."REGRNRATION BUFF", in2 := 85)
   END_RUNG wire#w1
   // the same network as SCL:
   "AUTO SUB OUTPUT"."SFV-1 – OPEN" := (("MFG PROCESS".MFG >= 7) AND ("MFG PROCESS".MFG < 20)) OR ("AlwaysTRUE" AND ("REGENRATION DB"."REGRNRATION BUFF" >= 65) AND ("REGENRATION DB"."REGRNRATION BUFF" < 85));
END_REGION

REGION Network 14: SFV-2 – OPEN
   RUNG wire#powerrail
      { S7_Templates := "SrcType := Int" } GE_Contact(in1 := "MFG PROCESS".MFG, in2 := 7)
      { S7_Templates := "SrcType := Int" } LT_Contact(in1 := "MFG PROCESS".MFG, in2 := 20)
      wire#w1
      Coil( "AUTO SUB OUTPUT"."SFV-2 – OPEN" )
   END_RUNG
   RUNG wire#powerrail
      { S7_Templates := "SrcType := Int" } GE_Contact(in1 := "REGENRATION DB"."REGRNRATION BUFF", in2 := 105)
   END_RUNG wire#w1
   // the same network as SCL:
   "AUTO SUB OUTPUT"."SFV-2 – OPEN" := (("MFG PROCESS".MFG >= 7) AND ("MFG PROCESS".MFG < 20)) OR ("REGENRATION DB"."REGRNRATION BUFF" >= 105);
END_REGION

REGION Network 15: SFV-3 – OPEN
   RUNG wire#powerrail
      Contact( "AlwaysTRUE" )
      { S7_Templates := "SrcType := Int" } GE_Contact(in1 := "REGENRATION DB"."REGRNRATION BUFF", in2 := 5)
      { S7_Templates := "SrcType := Int" } LT_Contact(in1 := "REGENRATION DB"."REGRNRATION BUFF", in2 := 25)
      Coil( "AUTO SUB OUTPUT"."SFV-3 – OPEN" )
   END_RUNG
   // the same network as SCL:
   "AUTO SUB OUTPUT"."SFV-3 – OPEN" := "AlwaysTRUE" AND ("REGENRATION DB"."REGRNRATION BUFF" >= 5) AND ("REGENRATION DB"."REGRNRATION BUFF" < 25);
END_REGION

REGION Network 16: SFV-4 – OPEN
   RUNG wire#powerrail
      Contact( "AlwaysTRUE" )
      { S7_Templates := "SrcType := Int" } GE_Contact(in1 := "REGENRATION DB"."REGRNRATION BUFF", in2 := 5)
      { S7_Templates := "SrcType := Int" } LT_Contact(in1 := "REGENRATION DB"."REGRNRATION BUFF", in2 := 25)
      Coil( "AUTO SUB OUTPUT"."SFV-4 – OPEN" )
   END_RUNG
   // the same network as SCL:
   "AUTO SUB OUTPUT"."SFV-4 – OPEN" := "AlwaysTRUE" AND ("REGENRATION DB"."REGRNRATION BUFF" >= 5) AND ("REGENRATION DB"."REGRNRATION BUFF" < 25);
END_REGION

REGION Network 17: SFV-5 – OPEN
   RUNG wire#powerrail
      Contact( "AlwaysTRUE" )
      wire#w1
      { S7_Templates := "SrcType := Int" } GE_Contact(in1 := "REGENRATION DB"."REGRNRATION BUFF", in2 := 20)
      { S7_Templates := "SrcType := Int" } LT_Contact(in1 := "REGENRATION DB"."REGRNRATION BUFF", in2 := 40)
      wire#w2
      Coil( "AUTO SUB OUTPUT"."SFV-5 – OPEN" )
   END_RUNG
   RUNG wire#w1
      { S7_Templates := "SrcType := Int" } GE_Contact(in1 := "REGENRATION DB"."REGRNRATION BUFF", in2 := 55)
      { S7_Templates := "SrcType := Int" } LT_Contact(in1 := "REGENRATION DB"."REGRNRATION BUFF", in2 := 85)
   END_RUNG wire#w2
   // the same network as SCL:
   "AUTO SUB OUTPUT"."SFV-5 – OPEN" := "AlwaysTRUE" AND ((("REGENRATION DB"."REGRNRATION BUFF" >= 20) AND ("REGENRATION DB"."REGRNRATION BUFF" < 40)) OR (("REGENRATION DB"."REGRNRATION BUFF" >= 55) AND ("REGENRATION DB"."REGRNRATION BUFF" < 85)));
END_REGION

REGION Network 18: SFV-6 – OPEN
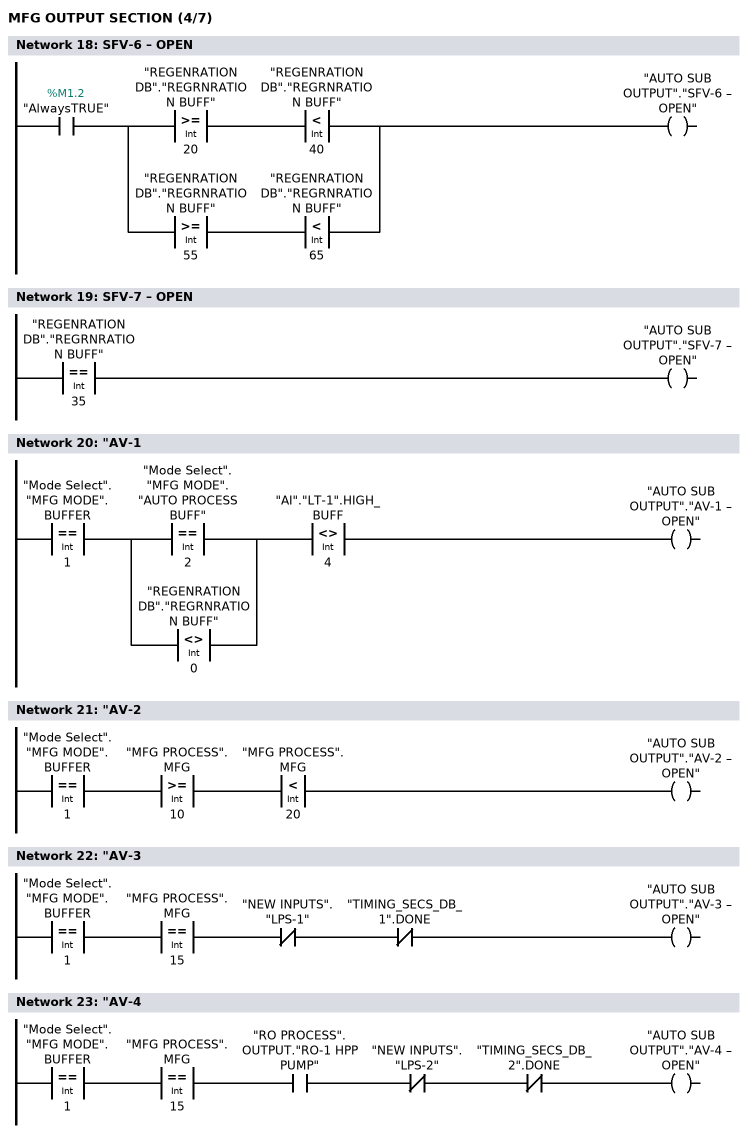
   RUNG wire#powerrail
      Contact( "AlwaysTRUE" )
      wire#w1
      { S7_Templates := "SrcType := Int" } GE_Contact(in1 := "REGENRATION DB"."REGRNRATION BUFF", in2 := 20)
      { S7_Templates := "SrcType := Int" } LT_Contact(in1 := "REGENRATION DB"."REGRNRATION BUFF", in2 := 40)
      wire#w2
      Coil( "AUTO SUB OUTPUT"."SFV-6 – OPEN" )
   END_RUNG
   RUNG wire#w1
      { S7_Templates := "SrcType := Int" } GE_Contact(in1 := "REGENRATION DB"."REGRNRATION BUFF", in2 := 55)
      { S7_Templates := "SrcType := Int" } LT_Contact(in1 := "REGENRATION DB"."REGRNRATION BUFF", in2 := 65)
   END_RUNG wire#w2
   // the same network as SCL:
   "AUTO SUB OUTPUT"."SFV-6 – OPEN" := "AlwaysTRUE" AND ((("REGENRATION DB"."REGRNRATION BUFF" >= 20) AND ("REGENRATION DB"."REGRNRATION BUFF" < 40)) OR (("REGENRATION DB"."REGRNRATION BUFF" >= 55) AND ("REGENRATION DB"."REGRNRATION BUFF" < 65)));
END_REGION

REGION Network 19: SFV-7 – OPEN
   RUNG wire#powerrail
      { S7_Templates := "SrcType := Int" } EQ_Contact(in1 := "REGENRATION DB"."REGRNRATION BUFF", in2 := 35)
      Coil( "AUTO SUB OUTPUT"."SFV-7 – OPEN" )
   END_RUNG
   // the same network as SCL:
   "AUTO SUB OUTPUT"."SFV-7 – OPEN" := "REGENRATION DB"."REGRNRATION BUFF" = 35;
END_REGION

REGION Network 20: "AV-1
   RUNG wire#powerrail
      { S7_Templates := "SrcType := Int" } EQ_Contact(in1 := "Mode Select"."MFG MODE".BUFFER, in2 := 1)
      wire#w1
      { S7_Templates := "SrcType := Int" } EQ_Contact(in1 := "Mode Select"."MFG MODE"."AUTO PROCESS BUFF", in2 := 2)
      wire#w2
      { S7_Templates := "SrcType := Int" } NE_Contact(in1 := "AI"."LT-1".HIGH_BUFF, in2 := 4)
      Coil( "AUTO SUB OUTPUT"."AV-1 – OPEN" )
   END_RUNG
   RUNG wire#w1
      { S7_Templates := "SrcType := Int" } NE_Contact(in1 := "REGENRATION DB"."REGRNRATION BUFF", in2 := 0)
   END_RUNG wire#w2
   // the same network as SCL:
   "AUTO SUB OUTPUT"."AV-1 – OPEN" := ("Mode Select"."MFG MODE".BUFFER = 1) AND (("Mode Select"."MFG MODE"."AUTO PROCESS BUFF" = 2) OR ("REGENRATION DB"."REGRNRATION BUFF" <> 0)) AND ("AI"."LT-1".HIGH_BUFF <> 4);
END_REGION

REGION Network 21: "AV-2
   RUNG wire#powerrail
      { S7_Templates := "SrcType := Int" } EQ_Contact(in1 := "Mode Select"."MFG MODE".BUFFER, in2 := 1)
      { S7_Templates := "SrcType := Int" } GE_Contact(in1 := "MFG PROCESS".MFG, in2 := 10)
      { S7_Templates := "SrcType := Int" } LT_Contact(in1 := "MFG PROCESS".MFG, in2 := 20)
      Coil( "AUTO SUB OUTPUT"."AV-2 – OPEN" )
   END_RUNG
   // the same network as SCL:
   "AUTO SUB OUTPUT"."AV-2 – OPEN" := ("Mode Select"."MFG MODE".BUFFER = 1) AND ("MFG PROCESS".MFG >= 10) AND ("MFG PROCESS".MFG < 20);
END_REGION

REGION Network 22: "AV-3
   RUNG wire#powerrail
      { S7_Templates := "SrcType := Int" } EQ_Contact(in1 := "Mode Select"."MFG MODE".BUFFER, in2 := 1)
      { S7_Templates := "SrcType := Int" } EQ_Contact(in1 := "MFG PROCESS".MFG, in2 := 15)
      I_Contact( "NEW INPUTS"."LPS-1" )
      I_Contact( "TIMING_SECS_DB_1".DONE )
      Coil( "AUTO SUB OUTPUT"."AV-3 – OPEN" )
   END_RUNG
   // the same network as SCL:
   "AUTO SUB OUTPUT"."AV-3 – OPEN" := ("Mode Select"."MFG MODE".BUFFER = 1) AND ("MFG PROCESS".MFG = 15) AND NOT "NEW INPUTS"."LPS-1" AND NOT "TIMING_SECS_DB_1".DONE;
END_REGION

REGION Network 23: "AV-4
   RUNG wire#powerrail
      { S7_Templates := "SrcType := Int" } EQ_Contact(in1 := "Mode Select"."MFG MODE".BUFFER, in2 := 1)
      { S7_Templates := "SrcType := Int" } EQ_Contact(in1 := "MFG PROCESS".MFG, in2 := 15)
      Contact( "RO PROCESS".OUTPUT."RO-1 HPP PUMP" )
      I_Contact( "NEW INPUTS"."LPS-2" )
      I_Contact( "TIMING_SECS_DB_2".DONE )
      Coil( "AUTO SUB OUTPUT"."AV-4 – OPEN" )
   END_RUNG
   // the same network as SCL:
   "AUTO SUB OUTPUT"."AV-4 – OPEN" := ("Mode Select"."MFG MODE".BUFFER = 1) AND ("MFG PROCESS".MFG = 15) AND "RO PROCESS".OUTPUT."RO-1 HPP PUMP" AND NOT "NEW INPUTS"."LPS-2" AND NOT "TIMING_SECS_DB_2".DONE;
END_REGION

REGION Network 24: DP-1
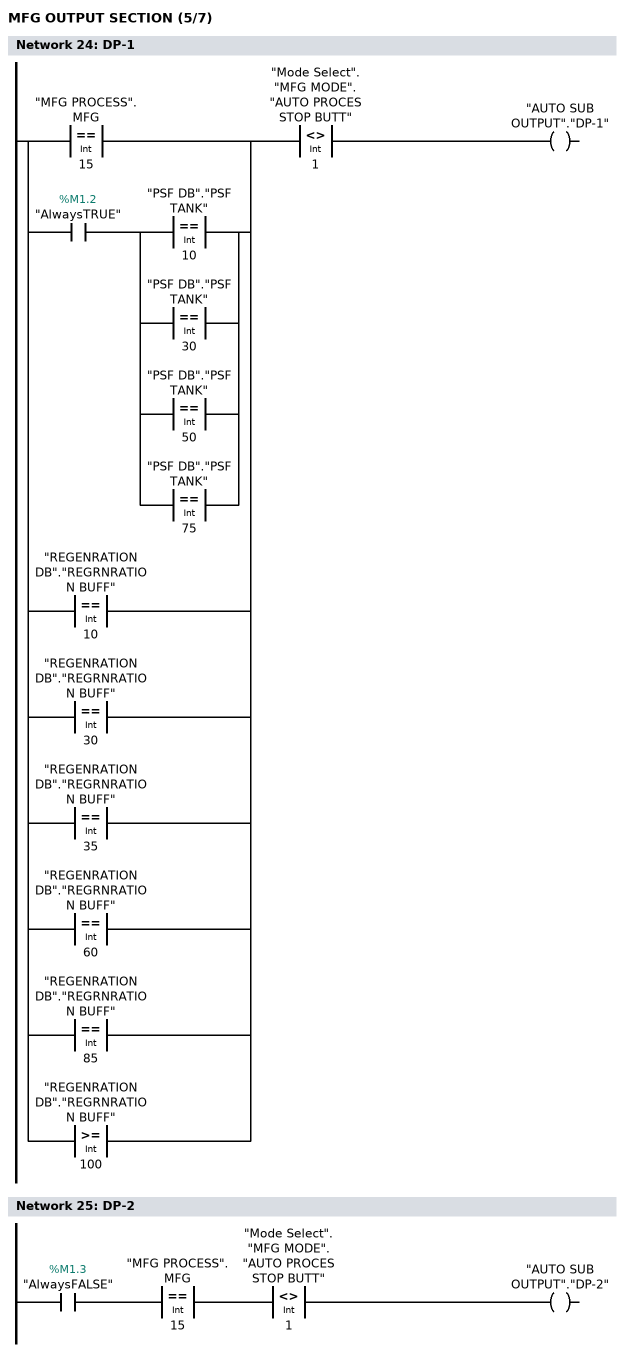
   RUNG wire#powerrail
      { S7_Templates := "SrcType := Int" } EQ_Contact(in1 := "MFG PROCESS".MFG, in2 := 15)
      wire#w1
      { S7_Templates := "SrcType := Int" } NE_Contact(in1 := "Mode Select"."MFG MODE"."AUTO PROCES STOP BUTT", in2 := 1)
      Coil( "AUTO SUB OUTPUT"."DP-1" )
   END_RUNG
   RUNG wire#powerrail
      Contact( "AlwaysTRUE" )
      wire#w2
      { S7_Templates := "SrcType := Int" } EQ_Contact(in1 := "PSF DB"."PSF TANK", in2 := 10)
   END_RUNG wire#w1
   RUNG wire#w2
      { S7_Templates := "SrcType := Int" } EQ_Contact(in1 := "PSF DB"."PSF TANK", in2 := 30)
   END_RUNG wire#w1
   RUNG wire#w2
      { S7_Templates := "SrcType := Int" } EQ_Contact(in1 := "PSF DB"."PSF TANK", in2 := 50)
   END_RUNG wire#w1
   RUNG wire#w2
      { S7_Templates := "SrcType := Int" } EQ_Contact(in1 := "PSF DB"."PSF TANK", in2 := 75)
   END_RUNG wire#w1
   RUNG wire#powerrail
      { S7_Templates := "SrcType := Int" } EQ_Contact(in1 := "REGENRATION DB"."REGRNRATION BUFF", in2 := 10)
   END_RUNG wire#w1
   RUNG wire#powerrail
      { S7_Templates := "SrcType := Int" } EQ_Contact(in1 := "REGENRATION DB"."REGRNRATION BUFF", in2 := 30)
   END_RUNG wire#w1
   RUNG wire#powerrail
      { S7_Templates := "SrcType := Int" } EQ_Contact(in1 := "REGENRATION DB"."REGRNRATION BUFF", in2 := 35)
   END_RUNG wire#w1
   RUNG wire#powerrail
      { S7_Templates := "SrcType := Int" } EQ_Contact(in1 := "REGENRATION DB"."REGRNRATION BUFF", in2 := 60)
   END_RUNG wire#w1
   RUNG wire#powerrail
      { S7_Templates := "SrcType := Int" } EQ_Contact(in1 := "REGENRATION DB"."REGRNRATION BUFF", in2 := 85)
   END_RUNG wire#w1
   RUNG wire#powerrail
      { S7_Templates := "SrcType := Int" } GE_Contact(in1 := "REGENRATION DB"."REGRNRATION BUFF", in2 := 100)
   END_RUNG wire#w1
   // the same network as SCL:
   "AUTO SUB OUTPUT"."DP-1" := (("MFG PROCESS".MFG = 15) OR ("AlwaysTRUE" AND (("PSF DB"."PSF TANK" = 10) OR ("PSF DB"."PSF TANK" = 30) OR ("PSF DB"."PSF TANK" = 50) OR ("PSF DB"."PSF TANK" = 75))) OR ("REGENRATION DB"."REGRNRATION BUFF" = 10) OR ("REGENRATION DB"."REGRNRATION BUFF" = 30) OR ("REGENRATION DB"."REGRNRATION BUFF" = 35) OR ("REGENRATION DB"."REGRNRATION BUFF" = 60) OR ("REGENRATION DB"."REGRNRATION BUFF" = 85) OR ("REGENRATION DB"."REGRNRATION BUFF" >= 100)) AND ("Mode Select"."MFG MODE"."AUTO PROCES STOP BUTT" <> 1);
END_REGION

REGION Network 25: DP-2
   RUNG wire#powerrail
      Contact( "AlwaysFALSE" )
      { S7_Templates := "SrcType := Int" } EQ_Contact(in1 := "MFG PROCESS".MFG, in2 := 15)
      { S7_Templates := "SrcType := Int" } NE_Contact(in1 := "Mode Select"."MFG MODE"."AUTO PROCES STOP BUTT", in2 := 1)
      Coil( "AUTO SUB OUTPUT"."DP-2" )
   END_RUNG
   // the same network as SCL:
   "AUTO SUB OUTPUT"."DP-2" := "AlwaysFALSE" AND ("MFG PROCESS".MFG = 15) AND ("Mode Select"."MFG MODE"."AUTO PROCES STOP BUTT" <> 1);
END_REGION

REGION Network 26: DP-3
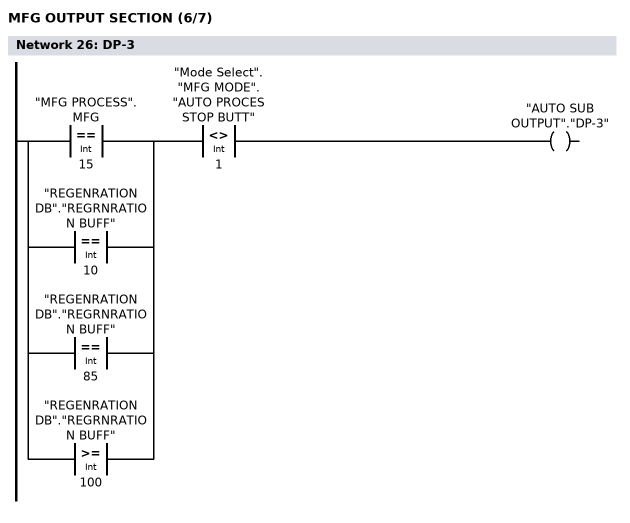
   RUNG wire#powerrail
      { S7_Templates := "SrcType := Int" } EQ_Contact(in1 := "MFG PROCESS".MFG, in2 := 15)
      wire#w1
      { S7_Templates := "SrcType := Int" } NE_Contact(in1 := "Mode Select"."MFG MODE"."AUTO PROCES STOP BUTT", in2 := 1)
      Coil( "AUTO SUB OUTPUT"."DP-3" )
   END_RUNG
   RUNG wire#powerrail
      { S7_Templates := "SrcType := Int" } EQ_Contact(in1 := "REGENRATION DB"."REGRNRATION BUFF", in2 := 10)
   END_RUNG wire#w1
   RUNG wire#powerrail
      { S7_Templates := "SrcType := Int" } EQ_Contact(in1 := "REGENRATION DB"."REGRNRATION BUFF", in2 := 85)
   END_RUNG wire#w1
   RUNG wire#powerrail
      { S7_Templates := "SrcType := Int" } GE_Contact(in1 := "REGENRATION DB"."REGRNRATION BUFF", in2 := 100)
   END_RUNG wire#w1
   // the same network as SCL:
   "AUTO SUB OUTPUT"."DP-3" := (("MFG PROCESS".MFG = 15) OR ("REGENRATION DB"."REGRNRATION BUFF" = 10) OR ("REGENRATION DB"."REGRNRATION BUFF" = 85) OR ("REGENRATION DB"."REGRNRATION BUFF" >= 100)) AND ("Mode Select"."MFG MODE"."AUTO PROCES STOP BUTT" <> 1);
END_REGION

REGION Network 27: FEED PUMP
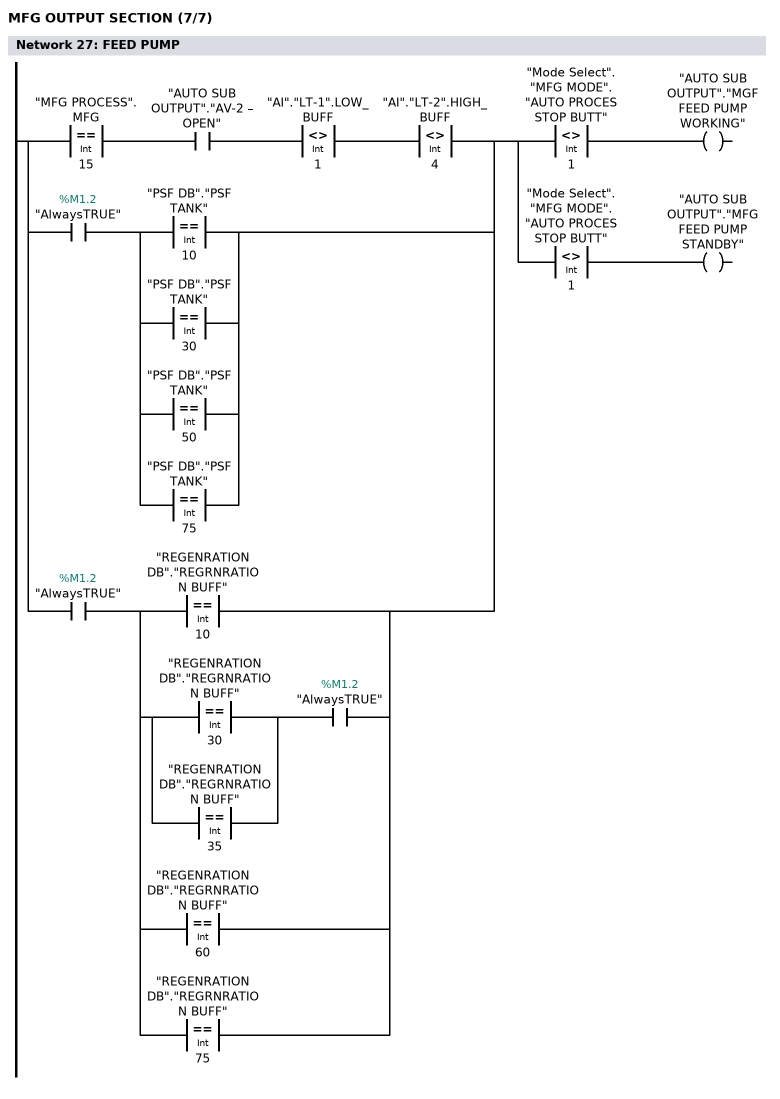
   RUNG wire#powerrail
      { S7_Templates := "SrcType := Int" } EQ_Contact(in1 := "MFG PROCESS".MFG, in2 := 15)
      Contact( "AUTO SUB OUTPUT"."AV-2 – OPEN" )
      { S7_Templates := "SrcType := Int" } NE_Contact(in1 := "AI"."LT-1".LOW_BUFF, in2 := 1)
      { S7_Templates := "SrcType := Int" } NE_Contact(in1 := "AI"."LT-2".HIGH_BUFF, in2 := 4)
      wire#w1
      { S7_Templates := "SrcType := Int" } NE_Contact(in1 := "Mode Select"."MFG MODE"."AUTO PROCES STOP BUTT", in2 := 1)
      Coil( "AUTO SUB OUTPUT"."MGF FEED PUMP WORKING" )
   END_RUNG
   RUNG wire#powerrail
      Contact( "AlwaysTRUE" )
      wire#w2
      { S7_Templates := "SrcType := Int" } EQ_Contact(in1 := "PSF DB"."PSF TANK", in2 := 10)
   END_RUNG wire#w1
   RUNG wire#w2
      { S7_Templates := "SrcType := Int" } EQ_Contact(in1 := "PSF DB"."PSF TANK", in2 := 30)
   END_RUNG wire#w1
   RUNG wire#w2
      { S7_Templates := "SrcType := Int" } EQ_Contact(in1 := "PSF DB"."PSF TANK", in2 := 50)
   END_RUNG wire#w1
   RUNG wire#w2
      { S7_Templates := "SrcType := Int" } EQ_Contact(in1 := "PSF DB"."PSF TANK", in2 := 75)
   END_RUNG wire#w1
   RUNG wire#powerrail
      Contact( "AlwaysTRUE" )
      wire#w3
      { S7_Templates := "SrcType := Int" } EQ_Contact(in1 := "REGENRATION DB"."REGRNRATION BUFF", in2 := 10)
   END_RUNG wire#w1
   RUNG wire#w3
      { S7_Templates := "SrcType := Int" } EQ_Contact(in1 := "REGENRATION DB"."REGRNRATION BUFF", in2 := 30)
      wire#w4
      Contact( "AlwaysTRUE" )
   END_RUNG wire#w1
   RUNG wire#w3
      { S7_Templates := "SrcType := Int" } EQ_Contact(in1 := "REGENRATION DB"."REGRNRATION BUFF", in2 := 35)
   END_RUNG wire#w4
   RUNG wire#w3
      { S7_Templates := "SrcType := Int" } EQ_Contact(in1 := "REGENRATION DB"."REGRNRATION BUFF", in2 := 60)
   END_RUNG wire#w1
   RUNG wire#w3
      { S7_Templates := "SrcType := Int" } EQ_Contact(in1 := "REGENRATION DB"."REGRNRATION BUFF", in2 := 75)
   END_RUNG wire#w1
   RUNG wire#w1
      { S7_Templates := "SrcType := Int" } NE_Contact(in1 := "Mode Select"."MFG MODE"."AUTO PROCES STOP BUTT", in2 := 1)
      Coil( "AUTO SUB OUTPUT"."MFG FEED PUMP STANDBY" )
   END_RUNG
   // the same network as SCL:
   #_w1 := (("MFG PROCESS".MFG = 15) AND "AUTO SUB OUTPUT"."AV-2 – OPEN" AND ("AI"."LT-1".LOW_BUFF <> 1) AND ("AI"."LT-2".HIGH_BUFF <> 4)) OR ("AlwaysTRUE" AND (("PSF DB"."PSF TANK" = 10) OR ("PSF DB"."PSF TANK" = 30) OR ("PSF DB"."PSF TANK" = 50) OR ("PSF DB"."PSF TANK" = 75))) OR ("AlwaysTRUE" AND (("REGENRATION DB"."REGRNRATION BUFF" = 10) OR ((("REGENRATION DB"."REGRNRATION BUFF" = 30) OR ("REGENRATION DB"."REGRNRATION BUFF" = 35)) AND "AlwaysTRUE") OR ("REGENRATION DB"."REGRNRATION BUFF" = 60) OR ("REGENRATION DB"."REGRNRATION BUFF" = 75)));
   "AUTO SUB OUTPUT"."MGF FEED PUMP WORKING" := #_w1 AND ("Mode Select"."MFG MODE"."AUTO PROCES STOP BUTT" <> 1);
   "AUTO SUB OUTPUT"."MFG FEED PUMP STANDBY" := #_w1 AND ("Mode Select"."MFG MODE"."AUTO PROCES STOP BUTT" <> 1);
END_REGION
END_FUNCTION

FUNCTION "REGENRATION PROCESS" : Void   // FC14, LAD
{ S7_Optimized_Access := 'TRUE' }
// stored: SetENOAutomatically false
BEGIN

REGION Network 2: START PROCESS
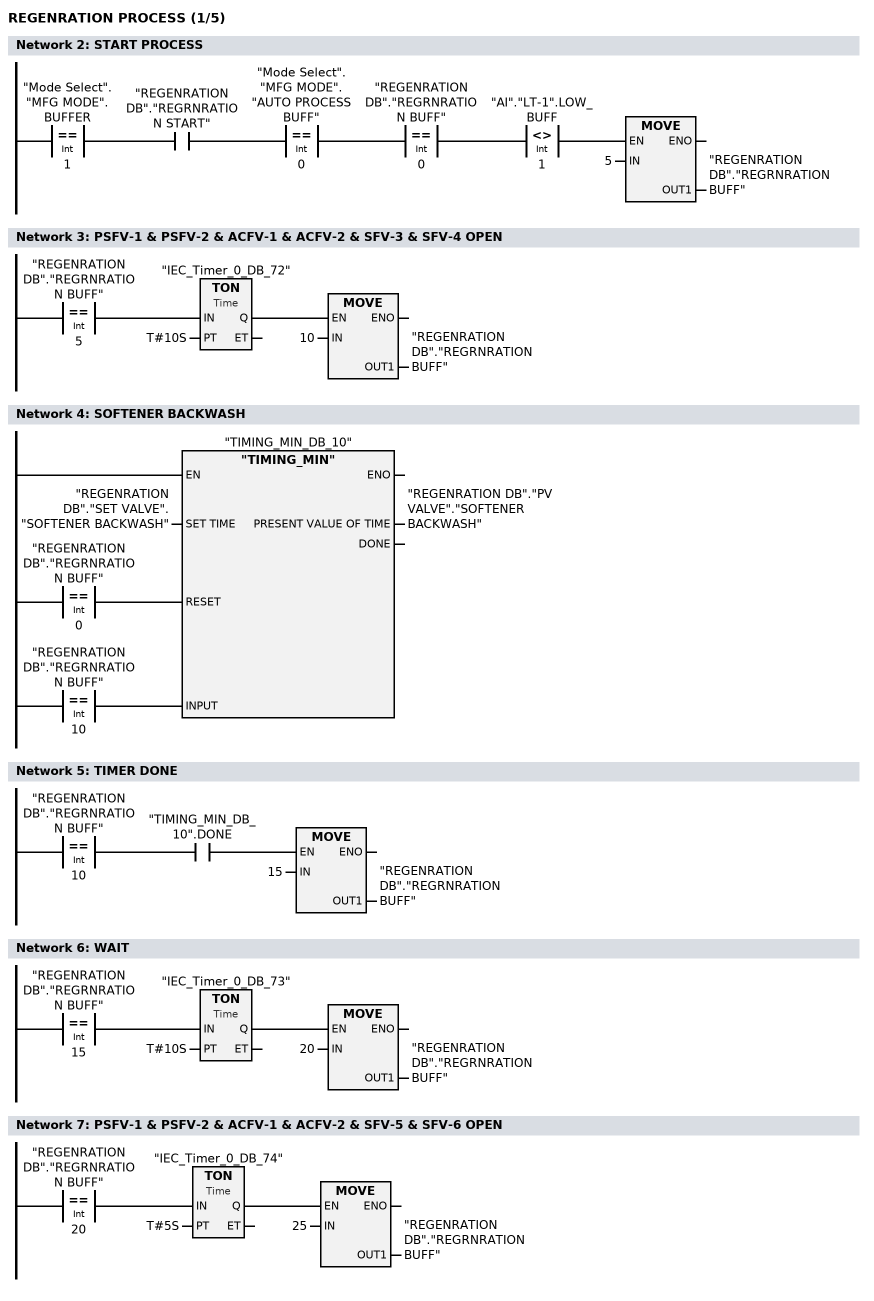
   RUNG wire#powerrail
      { S7_Templates := "SrcType := Int" } EQ_Contact(in1 := "Mode Select"."MFG MODE".BUFFER, in2 := 1)
      Contact( "REGENRATION DB"."REGRNRATION START" )
      { S7_Templates := "SrcType := Int" } EQ_Contact(in1 := "Mode Select"."MFG MODE"."AUTO PROCESS BUFF", in2 := 0)
      { S7_Templates := "SrcType := Int" } EQ_Contact(in1 := "REGENRATION DB"."REGRNRATION BUFF", in2 := 0)
      { S7_Templates := "SrcType := Int" } NE_Contact(in1 := "AI"."LT-1".LOW_BUFF, in2 := 1)
      Move(in := 5, out1 => "REGENRATION DB"."REGRNRATION BUFF")
   END_RUNG
   // the same network as SCL:
   IF ("Mode Select"."MFG MODE".BUFFER = 1) AND "REGENRATION DB"."REGRNRATION START" AND ("Mode Select"."MFG MODE"."AUTO PROCESS BUFF" = 0) AND ("REGENRATION DB"."REGRNRATION BUFF" = 0) AND ("AI"."LT-1".LOW_BUFF <> 1) THEN
       "REGENRATION DB"."REGRNRATION BUFF" := 5;
   END_IF;
END_REGION

REGION Network 3: PSFV-1 & PSFV-2 & ACFV-1 & ACFV-2 & SFV-3 & SFV-4 OPEN
   RUNG wire#powerrail
      { S7_Templates := "SrcType := Int" } EQ_Contact(in1 := "REGENRATION DB"."REGRNRATION BUFF", in2 := 5)
      { S7_Templates := "time_type := Time" } "IEC_Timer_0_DB_72".TON(pt := T#10S, et =>)
      Move(in := 10, out1 => "REGENRATION DB"."REGRNRATION BUFF")
   END_RUNG
   // the same network as SCL:
   "IEC_Timer_0_DB_72".TON(IN := "REGENRATION DB"."REGRNRATION BUFF" = 5, PT := T#10S);
   IF "IEC_Timer_0_DB_72".Q THEN "REGENRATION DB"."REGRNRATION BUFF" := 10; END_IF;
END_REGION

REGION Network 4: SOFTENER BACKWASH
   RUNG wire#powerrail
      "TIMING_MIN_DB_10"(RESET := wire#w1, INPUT := wire#w2, "SET TIME" := "REGENRATION DB"."SET VALVE"."SOFTENER BACKWASH", "PRESENT VALUE OF TIME" => "REGENRATION DB"."PV VALVE"."SOFTENER BACKWASH", DONE =>)
   END_RUNG
   RUNG wire#powerrail
      { S7_Templates := "SrcType := Int" } EQ_Contact(in1 := "REGENRATION DB"."REGRNRATION BUFF", in2 := 0)
   END_RUNG wire#w1
   RUNG wire#powerrail
      { S7_Templates := "SrcType := Int" } EQ_Contact(in1 := "REGENRATION DB"."REGRNRATION BUFF", in2 := 10)
   END_RUNG wire#w2
   // the same network as SCL:
   "TIMING_MIN_DB_10"("SET TIME" := "REGENRATION DB"."SET VALVE"."SOFTENER BACKWASH",   // "TIMING_MIN"
                      RESET := "REGENRATION DB"."REGRNRATION BUFF" = 0,
                      INPUT := "REGENRATION DB"."REGRNRATION BUFF" = 10,
                      "PRESENT VALUE OF TIME" => "REGENRATION DB"."PV VALVE"."SOFTENER BACKWASH");
END_REGION

REGION Network 5: TIMER DONE
   RUNG wire#powerrail
      { S7_Templates := "SrcType := Int" } EQ_Contact(in1 := "REGENRATION DB"."REGRNRATION BUFF", in2 := 10)
      Contact( "TIMING_MIN_DB_10".DONE )
      Move(in := 15, out1 => "REGENRATION DB"."REGRNRATION BUFF")
   END_RUNG
   // the same network as SCL:
   IF ("REGENRATION DB"."REGRNRATION BUFF" = 10) AND "TIMING_MIN_DB_10".DONE THEN
       "REGENRATION DB"."REGRNRATION BUFF" := 15;
   END_IF;
END_REGION

REGION Network 6: WAIT
   RUNG wire#powerrail
      { S7_Templates := "SrcType := Int" } EQ_Contact(in1 := "REGENRATION DB"."REGRNRATION BUFF", in2 := 15)
      { S7_Templates := "time_type := Time" } "IEC_Timer_0_DB_73".TON(pt := T#10S, et =>)
      Move(in := 20, out1 => "REGENRATION DB"."REGRNRATION BUFF")
   END_RUNG
   // the same network as SCL:
   "IEC_Timer_0_DB_73".TON(IN := "REGENRATION DB"."REGRNRATION BUFF" = 15, PT := T#10S);
   IF "IEC_Timer_0_DB_73".Q THEN "REGENRATION DB"."REGRNRATION BUFF" := 20; END_IF;
END_REGION

REGION Network 7: PSFV-1 & PSFV-2 & ACFV-1 & ACFV-2 & SFV-5 & SFV-6 OPEN
   RUNG wire#powerrail
      { S7_Templates := "SrcType := Int" } EQ_Contact(in1 := "REGENRATION DB"."REGRNRATION BUFF", in2 := 20)
      { S7_Templates := "time_type := Time" } "IEC_Timer_0_DB_74".TON(pt := T#5S, et =>)
      Move(in := 25, out1 => "REGENRATION DB"."REGRNRATION BUFF")
   END_RUNG
   // the same network as SCL:
   "IEC_Timer_0_DB_74".TON(IN := "REGENRATION DB"."REGRNRATION BUFF" = 20, PT := T#5S);
   IF "IEC_Timer_0_DB_74".Q THEN "REGENRATION DB"."REGRNRATION BUFF" := 25; END_IF;
END_REGION

REGION Network 8: SFV-3 & SFV-4 CLOSE
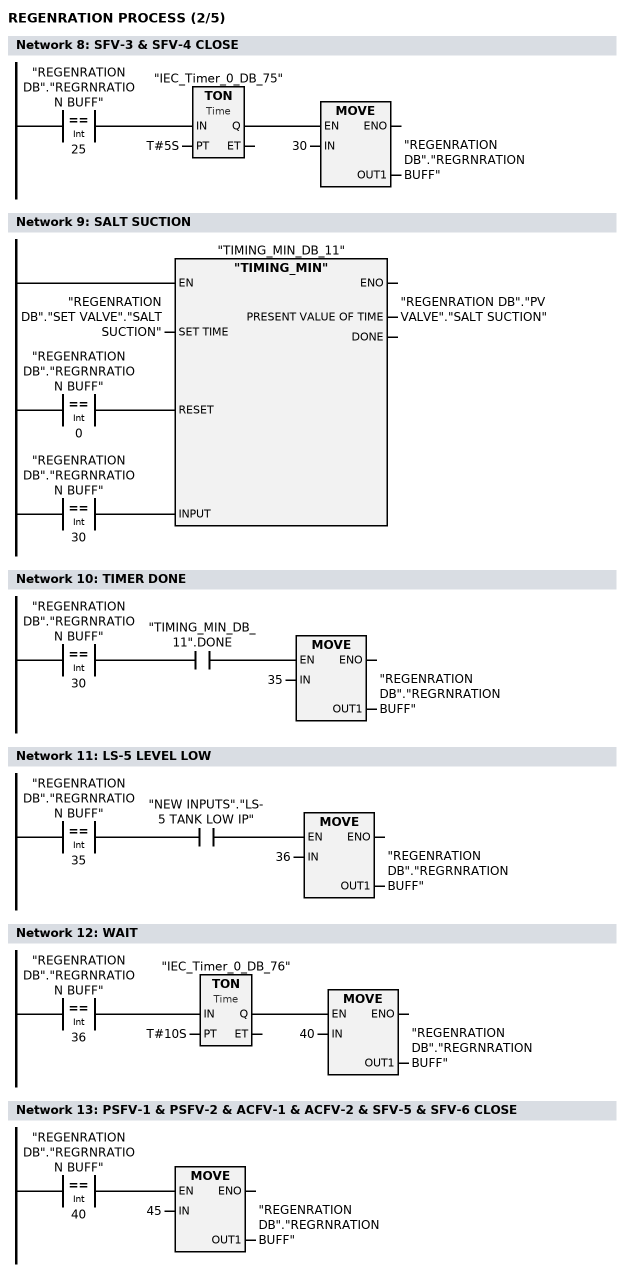
   RUNG wire#powerrail
      { S7_Templates := "SrcType := Int" } EQ_Contact(in1 := "REGENRATION DB"."REGRNRATION BUFF", in2 := 25)
      { S7_Templates := "time_type := Time" } "IEC_Timer_0_DB_75".TON(pt := T#5S, et =>)
      Move(in := 30, out1 => "REGENRATION DB"."REGRNRATION BUFF")
   END_RUNG
   // the same network as SCL:
   "IEC_Timer_0_DB_75".TON(IN := "REGENRATION DB"."REGRNRATION BUFF" = 25, PT := T#5S);
   IF "IEC_Timer_0_DB_75".Q THEN "REGENRATION DB"."REGRNRATION BUFF" := 30; END_IF;
END_REGION

REGION Network 9: SALT SUCTION
   RUNG wire#powerrail
      "TIMING_MIN_DB_11"(RESET := wire#w1, INPUT := wire#w2, "SET TIME" := "REGENRATION DB"."SET VALVE"."SALT SUCTION", "PRESENT VALUE OF TIME" => "REGENRATION DB"."PV VALVE"."SALT SUCTION", DONE =>)
   END_RUNG
   RUNG wire#powerrail
      { S7_Templates := "SrcType := Int" } EQ_Contact(in1 := "REGENRATION DB"."REGRNRATION BUFF", in2 := 0)
   END_RUNG wire#w1
   RUNG wire#powerrail
      { S7_Templates := "SrcType := Int" } EQ_Contact(in1 := "REGENRATION DB"."REGRNRATION BUFF", in2 := 30)
   END_RUNG wire#w2
   // the same network as SCL:
   "TIMING_MIN_DB_11"("SET TIME" := "REGENRATION DB"."SET VALVE"."SALT SUCTION",   // "TIMING_MIN"
                      RESET := "REGENRATION DB"."REGRNRATION BUFF" = 0,
                      INPUT := "REGENRATION DB"."REGRNRATION BUFF" = 30,
                      "PRESENT VALUE OF TIME" => "REGENRATION DB"."PV VALVE"."SALT SUCTION");
END_REGION

REGION Network 10: TIMER DONE
   RUNG wire#powerrail
      { S7_Templates := "SrcType := Int" } EQ_Contact(in1 := "REGENRATION DB"."REGRNRATION BUFF", in2 := 30)
      Contact( "TIMING_MIN_DB_11".DONE )
      Move(in := 35, out1 => "REGENRATION DB"."REGRNRATION BUFF")
   END_RUNG
   // the same network as SCL:
   IF ("REGENRATION DB"."REGRNRATION BUFF" = 30) AND "TIMING_MIN_DB_11".DONE THEN
       "REGENRATION DB"."REGRNRATION BUFF" := 35;
   END_IF;
END_REGION

REGION Network 11: LS-5 LEVEL LOW
   RUNG wire#powerrail
      { S7_Templates := "SrcType := Int" } EQ_Contact(in1 := "REGENRATION DB"."REGRNRATION BUFF", in2 := 35)
      Contact( "NEW INPUTS"."LS-5 TANK LOW IP" )
      Move(in := 36, out1 => "REGENRATION DB"."REGRNRATION BUFF")
   END_RUNG
   // the same network as SCL:
   IF ("REGENRATION DB"."REGRNRATION BUFF" = 35) AND "NEW INPUTS"."LS-5 TANK LOW IP" THEN
       "REGENRATION DB"."REGRNRATION BUFF" := 36;
   END_IF;
END_REGION

REGION Network 12: WAIT
   RUNG wire#powerrail
      { S7_Templates := "SrcType := Int" } EQ_Contact(in1 := "REGENRATION DB"."REGRNRATION BUFF", in2 := 36)
      { S7_Templates := "time_type := Time" } "IEC_Timer_0_DB_76".TON(pt := T#10S, et =>)
      Move(in := 40, out1 => "REGENRATION DB"."REGRNRATION BUFF")
   END_RUNG
   // the same network as SCL:
   "IEC_Timer_0_DB_76".TON(IN := "REGENRATION DB"."REGRNRATION BUFF" = 36, PT := T#10S);
   IF "IEC_Timer_0_DB_76".Q THEN "REGENRATION DB"."REGRNRATION BUFF" := 40; END_IF;
END_REGION

REGION Network 13: PSFV-1 & PSFV-2 & ACFV-1 & ACFV-2 & SFV-5 & SFV-6 CLOSE
   RUNG wire#powerrail
      { S7_Templates := "SrcType := Int" } EQ_Contact(in1 := "REGENRATION DB"."REGRNRATION BUFF", in2 := 40)
      Move(in := 45, out1 => "REGENRATION DB"."REGRNRATION BUFF")
   END_RUNG
   // the same network as SCL:
   IF "REGENRATION DB"."REGRNRATION BUFF" = 40 THEN "REGENRATION DB"."REGRNRATION BUFF" := 45; END_IF;
END_REGION

REGION Network 14: SALT HOLDING
